(* IEC 61131-3 sources: brOscatLib/oscatNetw (part 7) *)

(* ---- TN_INPUT_MENU_POPUP.st ---- *)
FUNCTION_BLOCK TN_INPUT_MENU_POPUP
    (*http://www.oscat.de/images/OSCATNetwork/oscat_netlib121_en.pdf#page=178*)
    (* sicherstellen das rechteck immer innerhalb screen positioniert wird *)

    IF (XUS_TN_MENU_POPUP.bo_Activ = FALSE) AND (XUS_TN_MENU_POPUP.bo_Create = TRUE) THEN
    	XUS_TN_MENU_POPUP.bo_Activ := TRUE;
    	XUS_TN_MENU_POPUP.bo_Create := FALSE;
    	XUS_TN_MENU_POPUP.bo_Destroy := FALSE;
    	XUS_TN_MENU_POPUP.bo_Update := TRUE;

      (* Sub-Menu-Texte *)

    	XUS_TN_MENU_POPUP.in_Menu_E_Count := ELEMENT_COUNT(SEP:=BYTE#35,ELEMENT:=XUS_TN_MENU_POPUP.st_Menu_Text);

    	(* Anzahl Zeilen (Sub-Menu-Texte) bestimmen *)
    	XUS_TN_MENU_POPUP.in_ROWS := XUS_TN_MENU_POPUP.in_Menu_E_Count;

    	(* längsten Sub-Menu-Text suchen *)
    	XUS_TN_MENU_POPUP.in_COLS := INT#00;

    	FOR in_Count := INT#01 TO XUS_TN_MENU_POPUP.in_ROWS DO;
    		XUS_TN_MENU_POPUP.in_COLS:=MAX(LEN(ELEMENT_GET(SEP:=BYTE#35,POS:=in_Count - 1,ELEMENT:=XUS_TN_MENU_POPUP.st_Menu_Text)),XUS_TN_MENU_POPUP.in_COLS);
    	END_FOR

    	(* Horizontale Position überprüfen und korrigieren *)
    	IF (XUS_TN_MENU_POPUP.in_X + XUS_TN_MENU_POPUP.in_COLS) > INT#75 THEN
    		XUS_TN_MENU_POPUP.in_X := INT#79 - XUS_TN_MENU_POPUP.in_COLS - INT#04;
    	END_IF

      (* Vertikale Position überprüfen und korrigieren *)
    	IF (XUS_TN_MENU_POPUP.in_Y + XUS_TN_MENU_POPUP.in_ROWS) > INT#21 THEN
    		XUS_TN_MENU_POPUP.in_Y := INT#23 - XUS_TN_MENU_POPUP.in_ROWS - INT#2;
    	END_IF

    	XUS_TN_SCREEN.bo_Modal_Dialog := TRUE;

    	(* Hintergrund sichern *)
    	FB_TN_SC_AREA_SAVE(	Iin_X1 := XUS_TN_MENU_POPUP.in_X,
    									Iin_Y1 := XUS_TN_MENU_POPUP.in_Y,
    									Iin_X2 := XUS_TN_MENU_POPUP.in_X + XUS_TN_MENU_POPUP.in_COLS + INT#04,
    									Iin_Y2 := XUS_TN_MENU_POPUP.in_Y + XUS_TN_MENU_POPUP.in_ROWS + INT#02,
    									XUS_TN_SCREEN := XUS_TN_SCREEN);

    	(* Rahmen für Submenu zeichnen *)
    	FB_TN_SC_BOX(	Iin_X1 := XUS_TN_MENU_POPUP.in_X,
    					Iin_Y1 := XUS_TN_MENU_POPUP.in_Y,
    					Iin_X2 := XUS_TN_MENU_POPUP.in_X + XUS_TN_MENU_POPUP.in_COLS + INT#03,
    					Iin_Y2 := XUS_TN_MENU_POPUP.in_Y + XUS_TN_MENU_POPUP.in_ROWS + INT#01,
    					Iby_FILL := BYTE#32, (* Füllung *)
    					Iin_BORDER := INT#01, (* Single-Line Border *)
    					Iby_ATTR := XUS_TN_MENU_POPUP.by_Attr_oF,
    					XUS_TN_SCREEN := XUS_TN_SCREEN);

    	(* Shadow für Submenu zeichnen *)
    	FB_TN_SC_ADD_SHADOW(Iin_X1 := XUS_TN_MENU_POPUP.in_X + INT#1,
    						Iin_Y1 := XUS_TN_MENU_POPUP.in_Y + INT#1,
    						Iin_X2 := XUS_TN_MENU_POPUP.in_X + XUS_TN_MENU_POPUP.in_COLS + INT#04,
    						Iin_Y2 := XUS_TN_MENU_POPUP.in_Y + XUS_TN_MENU_POPUP.in_ROWS + INT#02,
    						Iin_OPTION := INT#00,
    						XUS_TN_SCREEN := XUS_TN_SCREEN);

    	(* Parameter laden *)
    	in_COL := XUS_TN_MENU_POPUP.in_X;
    	in_ROW := XUS_TN_MENU_POPUP.in_Y;
    	in_ROWS := XUS_TN_MENU_POPUP.in_ROWS;
    	in_COLS := XUS_TN_MENU_POPUP.in_COLS;

    	(* Trennlinien zeichnen *)
    	in_COLS := in_COLS + INT#02; (* Text um 2 Zeichen verlängern *)

    	FOR in_Count := INT#01 TO XUS_TN_MENU_POPUP.in_Menu_E_Count DO;
    		in_ROW := in_ROW + INT#01;

    		IF ELEMENT_GET(SEP:=BYTE#35,POS:=in_Count - 1,ELEMENT:=XUS_TN_MENU_POPUP.st_Menu_Text) = '-' THEN

    			FB_TN_SC_LINE(	Iin_Y1 := in_ROW,
    							Iin_X1 := in_COL,
    							Iin_Y2 := in_ROW,
    							Iin_X2 := in_COL + in_COLS + INT#01,
    							Iby_ATTR := XUS_TN_MENU_POPUP.by_Attr_oF,
    							Iby_BORDER := BYTE#01,
    							XUS_TN_SCREEN := XUS_TN_SCREEN);
    		END_IF
    	END_FOR
    END_IF

    IF (XUS_TN_MENU_POPUP.bo_Activ = TRUE) THEN

    	CASE BYTE_TO_INT(XUS_TN_MENU_POPUP.by_Input_Exten_Code) OF

    	65: (* Cursor oben *)
    		in_Scroll_Offset := -1;
    		XUS_TN_MENU_POPUP.bo_Update := TRUE;

    	66: (* Cursor unten *)
    		in_Scroll_Offset := 1;
    		XUS_TN_MENU_POPUP.bo_Update := TRUE;

    	13:  (* Enter *)
    		XUS_TN_MENU_POPUP.bo_Destroy := TRUE;

    	27:  (* Escape*)
    		XUS_TN_MENU_POPUP.bo_Destroy := TRUE;
    		XUS_TN_MENU_POPUP.in_Cur_Item := INT#00;

    	67..68: (* Cursor links oder rechts *)
    		XUS_TN_MENU_POPUP.bo_Destroy := TRUE;
    		XUS_TN_MENU_POPUP.in_Cur_Item := INT#00;

    	END_CASE
    END_IF

    (* POPUP-Menu updaten *)
    IF (XUS_TN_MENU_POPUP.bo_Activ = TRUE) AND (XUS_TN_MENU_POPUP.bo_Update = TRUE) THEN

    	XUS_TN_MENU_POPUP.bo_Update := FALSE;

    	(* überprüfung + nächstes anwählbares Sub-Menu suchen *)
    	in_index := XUS_TN_MENU_POPUP.in_Cur_Item;

    	IF (in_index < INT#01) OR (in_index > XUS_TN_MENU_POPUP.in_Menu_E_Count) THEN
    		in_Scroll_Offset := INT#01;
    		in_index := XUS_TN_MENU_POPUP.in_Menu_E_Count;
    	END_IF

    	(* aktueller Index steht auf Trennzeichen -> ändern *)
    	IF ELEMENT_GET(SEP:=BYTE#35,POS:=in_index-1,ELEMENT:=XUS_TN_MENU_POPUP.st_Menu_Text) = '-' THEN
    		in_Scroll_Offset := INT#01;
    	END_IF

    	(* Scroll-Offset *)
    	IF in_Scroll_Offset <> INT#00 THEN

    		FOR in_Count := INT#01 TO XUS_TN_MENU_POPUP.in_Menu_E_Count DO;

    			in_index:=INC2(in_index,in_Scroll_Offset,1,XUS_TN_MENU_POPUP.in_Menu_E_Count);

    			IF ELEMENT_GET(SEP:=BYTE#35,POS:=in_index - 1,ELEMENT:=XUS_TN_MENU_POPUP.st_Menu_Text) <> '-' THEN
    				EXIT;
    			END_IF

    		END_FOR
    	END_IF

    	XUS_TN_MENU_POPUP.in_Cur_Item := in_index;
    	in_Scroll_Offset := INT#00;

    	(* Parameter laden *)
    	in_COL  := XUS_TN_MENU_POPUP.in_X;
    	in_ROW  := XUS_TN_MENU_POPUP.in_Y;
    	in_ROWS := XUS_TN_MENU_POPUP.in_ROWS;
    	in_COLS := XUS_TN_MENU_POPUP.in_COLS;

    	(* SUB-MENU-Titel ausgeben *)
    	in_COLS := in_COLS + INT#02; (* Text um 2 Zeichen verlängern *)

    	FOR in_Count := INT#01 TO XUS_TN_MENU_POPUP.in_Menu_E_Count DO;

    		in_ROW := in_ROW + INT#01;

    		(* Zeichenfarbe bestimmen *)
    		IF in_Count = XUS_TN_MENU_POPUP.in_Cur_Item THEN
    			by_ATTR := XUS_TN_MENU_POPUP.by_Attr_mF;
    		ELSE
    			by_ATTR := XUS_TN_MENU_POPUP.by_Attr_oF;
    		END_IF

    		FB_TN_SC_WRITE_C.Ist_STRING := ELEMENT_GET(SEP:=BYTE#35,POS:=in_Count - 1,ELEMENT:=XUS_TN_MENU_POPUP.st_Menu_Text);

    		IF FB_TN_SC_WRITE_C.Ist_STRING <> '-' THEN

    			FB_TN_SC_WRITE_C(	Iin_Y := in_ROW,
    								Iin_X := in_COL + INT#01,
    								Iby_ATTR := by_ATTR,
    								Iin_LENGTH := in_COLS,
    								Iin_OPTION := INT#02, (* Center *)
    								XUS_TN_SCREEN := XUS_TN_SCREEN);
    		END_IF
    	END_FOR
    END_IF

    (* POPUP-Menu entfernen (Destroy) *)
    IF (XUS_TN_MENU_POPUP.bo_Activ = TRUE) AND (XUS_TN_MENU_POPUP.bo_Destroy = TRUE) THEN

    	XUS_TN_MENU_POPUP.bo_Destroy := FALSE;
    	XUS_TN_MENU_POPUP.bo_Activ := FALSE;

    	(* alten Hintergrund aus Speicher wiederherstellen *)
    	FB_TN_SC_AREA_RESTORE(XUS_TN_SCREEN := XUS_TN_SCREEN);

    	XUS_TN_SCREEN.bo_Modal_Dialog := FALSE;
    END_IF

    (* revision history

    ks	06. apr. 2011	rev 1.1
    	list_len und list_get durch element_count und element_get ersetzt

    ks	10. mai. 2010	rev 1.0
    	original version
    *)
END_FUNCTION_BLOCK

(* ---- TN_INPUT_SELECT_POPUP.st ---- *)
FUNCTION_BLOCK TN_INPUT_SELECT_POPUP
    (*http://www.oscat.de/images/OSCATNetwork/oscat_netlib121_en.pdf#page=178*)
    (* Benutzereingabe auswerten -> Selektion Text n *)
    IF (XUS_TN_INPUT_CONTROL_DATA.bo_Focus = TRUE) THEN

    	by_Cur_Key := XUS_TN_INPUT_CONTROL_DATA.by_Input_Exten_Code;

    	IF (us_TN_MENU_POPUP.bo_Activ = FALSE) THEN
    		us_TN_MENU_POPUP.by_Input_Exten_Code := BYTE#00;

    		(* Return-Taste auswerten *)
    		IF (by_Cur_Key = BYTE#13) THEN
    			(* Popup-Menu parameter übergeben *)
    			us_TN_MENU_POPUP.in_Y := XUS_TN_INPUT_CONTROL_DATA.in_Y;
    			us_TN_MENU_POPUP.in_X := XUS_TN_INPUT_CONTROL_DATA.in_X;
    			us_TN_MENU_POPUP.by_Attr_mF := XUS_TN_INPUT_CONTROL_DATA.by_Attr_mF;
    			us_TN_MENU_POPUP.by_Attr_oF := XUS_TN_INPUT_CONTROL_DATA.by_Attr_oF;
    			us_TN_MENU_POPUP.st_Menu_Text := XUS_TN_INPUT_CONTROL_DATA.st_Input_Data;
    			us_TN_MENU_POPUP.bo_Create := TRUE;
    			us_TN_MENU_POPUP.in_Cur_Item := INT#00;
    		END_IF

    		IF (us_TN_MENU_POPUP.in_Cur_Item > INT#00) THEN
    			XUS_TN_INPUT_CONTROL_DATA.in_selected := us_TN_MENU_POPUP.in_Cur_Item;
    			XUS_TN_INPUT_CONTROL_DATA.bo_Input_Entered := TRUE;
    			XUS_TN_INPUT_CONTROL_DATA.bo_Update_Input := TRUE;
    			us_TN_MENU_POPUP.in_Cur_Item := INT#00;
    		END_IF

    	ELSE
    		us_TN_MENU_POPUP.by_Input_Exten_Code := by_Cur_Key;
    	END_IF

    	(* Popup-Menu zyklisch aufrufen *)
    	FB_TN_INPUT_MENU_POPUP(Xus_TN_MENU_POPUP := us_TN_MENU_POPUP, XUS_TN_SCREEN := XUS_TN_SCREEN);

    END_IF

    (* Aktualisierung der Anzeige *)
    IF (XUS_TN_INPUT_CONTROL_DATA.bo_Update_Input = TRUE) OR (XUS_TN_INPUT_CONTROL_DATA.bo_Update_All = TRUE) THEN

    	(* Title-Text ausgeben *)
    	IF XUS_TN_INPUT_CONTROL_DATA.bo_Update_All = TRUE THEN

    		IF (XUS_TN_INPUT_CONTROL_DATA.in_Title_X_Offset = INT#00) AND (XUS_TN_INPUT_CONTROL_DATA.in_Title_Y_Offset = INT#00) THEN
    			(* wenn Offset X,Y =0 dann Titlestring links vom Element positionieren *)
    			FB_TN_SC_WRITE.Iin_Y := XUS_TN_INPUT_CONTROL_DATA.in_Y;
    			FB_TN_SC_WRITE.Iin_X := XUS_TN_INPUT_CONTROL_DATA.in_X - LEN(XUS_TN_INPUT_CONTROL_DATA.st_Title_String);

    		ELSE
    			(* Title-Text durch Row, Color-Offset ausgeben *)
    			FB_TN_SC_WRITE.Iin_Y := XUS_TN_INPUT_CONTROL_DATA.in_Y + XUS_TN_INPUT_CONTROL_DATA.in_Title_Y_Offset;
    			FB_TN_SC_WRITE.Iin_X := XUS_TN_INPUT_CONTROL_DATA.in_X + XUS_TN_INPUT_CONTROL_DATA.in_Title_X_Offset;
    		END_IF

    		(* Title-Text durch Row, Color-Offset ausgeben *)
    		FB_TN_SC_WRITE(	Iby_ATTR := XUS_TN_INPUT_CONTROL_DATA.by_Title_Attr,
    						Ist_STRING := XUS_TN_INPUT_CONTROL_DATA.st_Title_String,
    						XUS_TN_SCREEN := XUS_TN_SCREEN);
    	END_IF

    	in_Element_Count := ELEMENT_COUNT(SEP:=BYTE#35,ELEMENT:=XUS_TN_INPUT_CONTROL_DATA.st_Input_Data);

    	IF in_Element_Count > INT#00 THEN

    		XUS_TN_INPUT_CONTROL_DATA.in_selected:=LIMIT(1,XUS_TN_INPUT_CONTROL_DATA.in_selected,in_Element_Count);

    		in_index := XUS_TN_INPUT_CONTROL_DATA.in_selected;

    		st_String := ELEMENT_GET(SEP:=BYTE#35,POS:=in_index - 1,ELEMENT:=XUS_TN_INPUT_CONTROL_DATA.st_Input_Data);

    		st_String:= FIX(str:=st_String,
    						L:=LEN(XUS_TN_INPUT_CONTROL_DATA.st_Input_Mask),
    						C:=BYTE#32,
    						M:=XUS_TN_INPUT_CONTROL_DATA.in_Input_Option);

    		XUS_TN_INPUT_CONTROL_DATA.st_Input_String := st_String;

    		IF XUS_TN_INPUT_CONTROL_DATA.bo_Focus = TRUE THEN
    			by_Attr := XUS_TN_INPUT_CONTROL_DATA.by_Attr_mF;
    		ELSE
    			by_Attr := XUS_TN_INPUT_CONTROL_DATA.by_Attr_oF;
    		END_IF

    		FB_TN_SC_WRITE(	Iin_X := XUS_TN_INPUT_CONTROL_DATA.in_X,
    								Iin_Y := XUS_TN_INPUT_CONTROL_DATA.in_Y,
    								Iby_ATTR := by_Attr,
    								Ist_STRING := st_String,
    								XUS_TN_SCREEN := XUS_TN_SCREEN );
    	END_IF

    	(* Cursor auf aktuelle Position setzen *)
    	XUS_TN_INPUT_CONTROL_DATA.in_Cursor_X := XUS_TN_INPUT_CONTROL_DATA.in_X;
    	XUS_TN_INPUT_CONTROL_DATA.in_Cursor_Y := XUS_TN_INPUT_CONTROL_DATA.in_Y;

    	(* Update-Flag's rücksetzen *)
    	XUS_TN_INPUT_CONTROL_DATA.bo_Update_All   := FALSE;
    	XUS_TN_INPUT_CONTROL_DATA.bo_Update_Input := FALSE;

    END_IF

    (* revision history

    ks	06. apr. 2011	rev 1.1
    	list_len und list_get durch element_count und element_get ersetzt

    ks	10. mai. 2010	rev 1.0
    	original version
    *)
END_FUNCTION_BLOCK

(* ---- TN_INPUT_SELECT_TEXT.st ---- *)
FUNCTION_BLOCK TN_INPUT_SELECT_TEXT
    (*http://www.oscat.de/images/OSCATNetwork/oscat_netlib121_en.pdf#page=180*)
    (* Benutzereingabe auswerten -> Selektion Text n *)
    IF XUS_TN_INPUT_CONTROL_DATA.bo_Focus = TRUE THEN

    (* Leertaste-Taste auswerten *)
    	IF XUS_TN_INPUT_CONTROL_DATA.by_Input_ASCII_Code = BYTE#32 THEN
    		XUS_TN_INPUT_CONTROL_DATA.in_selected := XUS_TN_INPUT_CONTROL_DATA.in_selected + INT#01;
    		XUS_TN_INPUT_CONTROL_DATA.bo_Update_Input := TRUE;
    	END_IF

    	(* Return-Taste auswerten *)
    	IF XUS_TN_INPUT_CONTROL_DATA.by_Input_Exten_Code = BYTE#13 THEN
    		XUS_TN_INPUT_CONTROL_DATA.bo_Input_Entered := TRUE;
    	END_IF

    END_IF

    (* Aktualisierung der Anzeige *)
    IF (XUS_TN_INPUT_CONTROL_DATA.bo_Update_Input = TRUE) OR (XUS_TN_INPUT_CONTROL_DATA.bo_Update_All = TRUE) THEN

    	(* Title-Text ausgeben *)
    	IF XUS_TN_INPUT_CONTROL_DATA.bo_Update_All = TRUE THEN

    		IF (XUS_TN_INPUT_CONTROL_DATA.in_Title_X_Offset = INT#00) AND (XUS_TN_INPUT_CONTROL_DATA.in_Title_Y_Offset = INT#00) THEN
    			(* wenn Offset X,Y =0 dann Titlestring links vom Element positionieren *)
    			FB_TN_SC_WRITE.Iin_Y := XUS_TN_INPUT_CONTROL_DATA.in_Y;
    			FB_TN_SC_WRITE.Iin_X := XUS_TN_INPUT_CONTROL_DATA.in_X - LEN(XUS_TN_INPUT_CONTROL_DATA.st_Title_String);

    		ELSE
    			(* Title-Text durch Row, Color-Offset ausgeben *)
    			FB_TN_SC_WRITE.Iin_Y := XUS_TN_INPUT_CONTROL_DATA.in_Y + XUS_TN_INPUT_CONTROL_DATA.in_Title_Y_Offset;
    			FB_TN_SC_WRITE.Iin_X := XUS_TN_INPUT_CONTROL_DATA.in_X + XUS_TN_INPUT_CONTROL_DATA.in_Title_X_Offset;
    		END_IF

    		(* Title-Text durch Row, Color-Offset ausgeben *)
    		FB_TN_SC_WRITE(	Iby_ATTR := XUS_TN_INPUT_CONTROL_DATA.by_Title_Attr,
    						Ist_STRING := XUS_TN_INPUT_CONTROL_DATA.st_Title_String,
    						XUS_TN_SCREEN := XUS_TN_SCREEN);

    	END_IF

    	(* Eingabezeile verarbeiten *)

    	(* Anzahl der Elemente bestimmen *)
    	in_count := ELEMENT_COUNT(SEP:=BYTE#35,ELEMENT:=XUS_TN_INPUT_CONTROL_DATA.st_Input_Data);

    	IF in_count > INT#00 THEN

    		IF XUS_TN_INPUT_CONTROL_DATA.in_selected < INT#1 THEN
    			XUS_TN_INPUT_CONTROL_DATA.in_selected := INT#01;
    		END_IF

    		IF XUS_TN_INPUT_CONTROL_DATA.in_selected > in_count THEN
    			XUS_TN_INPUT_CONTROL_DATA.in_selected := INT#01;
    		END_IF

    		st_String := ELEMENT_GET(SEP:=BYTE#35,POS:=XUS_TN_INPUT_CONTROL_DATA.in_selected - 1,ELEMENT:=XUS_TN_INPUT_CONTROL_DATA.st_Input_Data);

    		st_String := FIX(	str:=st_String,
    							L:=LEN(XUS_TN_INPUT_CONTROL_DATA.st_Input_Mask),
    							C:=BYTE#32,
    							M:=XUS_TN_INPUT_CONTROL_DATA.in_Input_Option);

    		XUS_TN_INPUT_CONTROL_DATA.st_Input_String := st_String;

    		IF XUS_TN_INPUT_CONTROL_DATA.bo_Focus = TRUE THEN
    			by_Attr := XUS_TN_INPUT_CONTROL_DATA.by_Attr_mF;
    		ELSE
    			by_Attr := XUS_TN_INPUT_CONTROL_DATA.by_Attr_oF;
    		END_IF

    		FB_TN_SC_WRITE(	Iin_Y := XUS_TN_INPUT_CONTROL_DATA.in_Y,
    						Iin_X := XUS_TN_INPUT_CONTROL_DATA.in_X,
    						Iby_ATTR := by_Attr,
    						Ist_STRING := st_String,
    						XUS_TN_SCREEN := XUS_TN_SCREEN);
    	END_IF

    	(* Cursor auf aktuelle Position setzen *)
    	XUS_TN_INPUT_CONTROL_DATA.in_Cursor_Y := XUS_TN_INPUT_CONTROL_DATA.in_Y;
    	XUS_TN_INPUT_CONTROL_DATA.in_Cursor_X := XUS_TN_INPUT_CONTROL_DATA.in_X;

    	(* Update-Flag's rücksetzen *)
    	XUS_TN_INPUT_CONTROL_DATA.bo_Update_All := FALSE;
    	XUS_TN_INPUT_CONTROL_DATA.bo_Update_Input := FALSE;

    END_IF

    (* revision history

    ks	06. apr. 2011	rev 1.1
    	list_len und list_get durch element_count und element_get ersetzt

    ks	10. mai. 2010	rev 1.0
    	original version
    *)
END_FUNCTION_BLOCK

(* ---- TN_RECEIVE.st ---- *)
FUNCTION_BLOCK TN_RECEIVE
    (*http://www.oscat.de/images/OSCATNetwork/oscat_netlib121_en.pdf#page=182*)
    (* Datenempfang auswertung *)
    XUS_TN_SCREEN.by_Input_ASCII_Code := BYTE#00;
    XUS_TN_SCREEN.by_Input_Exten_Code := BYTE#00;

    IF R_BUF.SIZE > UINT#0 THEN
    	(* empfangene Daten auswerten *)
    	REQ_Size := R_BUF.SIZE;
    	REQ1 := R_BUF.BUFFER[0];
    	REQ2 := R_BUF.BUFFER[1];
    	REQ3 := R_BUF.BUFFER[2];

    	IF REQ1 = BYTE#27 AND REQ_Size >= UINT#3 THEN (* Escape *)
    		IF REQ2 = BYTE#91 THEN (* Cursor code *)
    			IF (REQ3 >= BYTE#65 AND REQ3 <= BYTE#68) OR (REQ3 = BYTE#72) OR (REQ3 = BYTE#75) THEN (* 65..68 = Cursor o,u,r,l / 72 = POS1 / 75 = ENDE *)
    				XUS_TN_SCREEN.by_Input_Exten_Code := REQ3;
    			END_IF
    		ELSIF REQ2 = BYTE#79 THEN (* Sondertasten F1/F2/F3/F4 *)
    			IF REQ3 >= BYTE#80 AND REQ3 <= BYTE#83 THEN
    				XUS_TN_SCREEN.by_Input_Exten_Code := REQ3;
    			END_IF
    		END_IF
    	ELSIF REQ1 >= BYTE#32 AND REQ1 <= BYTE#126 THEN
    		XUS_TN_SCREEN.by_Input_ASCII_Code := REQ1;
    		XUS_TN_SCREEN.bo_Input_ASCII_IsNum := ISC_NUM(REQ1); (* Auswertung auf Zahleneingabe *)
    	ELSIF REQ1 = BYTE#8 OR REQ1 = BYTE#9 OR REQ1 = BYTE#13 OR REQ1 = BYTE#27 THEN (* prüfe auf Steuerzeichen 8=Backspace / 9=Tabulator / 13=Return / 27=Escape *)
    		XUS_TN_SCREEN.by_Input_Exten_Code := REQ1;
    	END_IF

    	(* Empfangsbuffer Datenlänge null eintragen (Telegramm zerstören *)
    	R_BUF.SIZE := UINT#00;
    END_IF

    (* revision history
    ks	10. mai. 2010	rev 1.0
    	original version
    *)
END_FUNCTION_BLOCK

(* ---- TN_SC_ADD_SHADOW.st ---- *)
FUNCTION_BLOCK TN_SC_ADD_SHADOW
    (*http://www.oscat.de/images/OSCATNetwork/oscat_netlib121_en.pdf#page=184*)
    IF TN_SC_XY2_ERROR(IIN_X1,IIN_Y1,IIN_X2,IIN_Y2) THEN RETURN; END_IF

    IF IIN_Y1 < 0 OR IIN_X1 < 0 OR IIN_Y2 < 0 OR IIN_X2 < 0 THEN RETURN; END_IF (* min werte prüfen *)
    IF IIN_Y1 > 23 OR IIN_X1 > 79 OR IIN_Y2 > 23 OR IIN_X2 > 79 THEN RETURN; END_IF (* max werte prüfen *)

    in_Offset := (IIN_Y1 * 80) + IIN_X2;

    IF IIN_OPTION = INT#00 THEN
    	(* Schatten durch Farbanpassung erzeugen *)
    	FOR in_Y := IIN_Y1 TO IIN_Y2 DO
    		XUS_TN_SCREEN.bya_COLOR[in_Offset] := TN_SC_SHADOW_ATTR(XUS_TN_SCREEN.bya_COLOR[in_Offset]);
    		in_Offset := in_Offset + 80;
    		XUS_TN_SCREEN.bya_Line_Update[in_Y] := TRUE; (* Zeile für Update eintragen *)
    	END_FOR
    ELSE
    	(* Schatten durch Farbe Schwarz und Leerzeichen erzeugen *)
    	FOR in_Y := IIN_Y1 TO IIN_Y2 DO
    		XUS_TN_SCREEN.bya_COLOR[in_Offset] := BYTE#00;
    		XUS_TN_SCREEN.bya_CHAR[in_Offset] := BYTE#32;
    		in_Offset := in_Offset + 80;
    		XUS_TN_SCREEN.bya_Line_Update[in_Y] := TRUE; (* Zeile für Update eintragen *)
    	END_FOR
    END_IF

    in_Offset := (IIN_Y2 * 80) + IIN_X1;

    IF IIN_OPTION = INT#00 THEN
    	(* Schatten durch Farbanpassung erzeugen *)
    	FOR in_X  := IIN_X1 TO IIN_X2 DO
    		XUS_TN_SCREEN.bya_COLOR[in_Offset] := TN_SC_SHADOW_ATTR(XUS_TN_SCREEN.bya_COLOR[in_Offset]);
    		in_Offset := in_Offset + 1;
    	END_FOR
    ELSE
    	(* Schatten durch Farbe Schwarz und Leerzeichen erzeugen *)
    	FOR in_X  := IIN_X1 TO IIN_X2 DO
    		XUS_TN_SCREEN.bya_COLOR[in_Offset] := BYTE#00;
    		XUS_TN_SCREEN.bya_CHAR[in_Offset] := BYTE#32;
    		in_Offset := in_Offset + 1;
    	END_FOR
    END_IF

    (* revision history
    ks	10. mai. 2010	rev 1.0
    	original version
    *)
END_FUNCTION_BLOCK

(* ---- TN_SC_AREA_RESTORE.st ---- *)
FUNCTION_BLOCK TN_SC_AREA_RESTORE
    (*http://www.oscat.de/images/OSCATNetwork/oscat_netlib121_en.pdf#page=184*)
    IF XUS_TN_SCREEN.bya_BACKUP[0] > BYTE#00 THEN

    	(* Parameter auslesen *)
    	in_X1 := BYTE_TO_INT(XUS_TN_SCREEN.bya_BACKUP[1]);
    	in_Y1 := BYTE_TO_INT(XUS_TN_SCREEN.bya_BACKUP[2]);
    	in_X2 := BYTE_TO_INT(XUS_TN_SCREEN.bya_BACKUP[3]);
    	in_Y2 := BYTE_TO_INT(XUS_TN_SCREEN.bya_BACKUP[4]);

    	IF TN_SC_XY2_ERROR(in_X1,in_Y1,in_X2,in_Y2) THEN RETURN; END_IF
    	in_Offset_2 := 5;

    	(* CHAR und COLOR von BUFFER wiederherstellen *)
    	FOR in_Y := in_Y1 TO in_Y2 DO

    		XUS_TN_SCREEN.bya_Line_Update[in_Y] := TRUE; (* Zeile zum Updaten freigeben *)
    		in_Offset_1 := (in_Y * 80) + in_X1;

    		FOR in_X := in_X1 TO in_X2 DO

    			XUS_TN_SCREEN.bya_CHAR[in_Offset_1] := XUS_TN_SCREEN.bya_BACKUP[in_Offset_2];
    			in_Offset_2 := in_Offset_2 + INT#01;

    			XUS_TN_SCREEN.bya_COLOR[in_Offset_1] := XUS_TN_SCREEN.bya_BACKUP[in_Offset_2];
    			in_Offset_2 := in_Offset_2 + INT#01;
    			in_Offset_1 := in_Offset_1 + INT#01;

    		END_FOR
    	END_FOR

    	(* Daten als ungültig markieren *)
    	XUS_TN_SCREEN.bya_BACKUP[0] := BYTE#00;
    END_IF

    (* revision history
    ks	10. mai. 2010	rev 1.0
    	original version
    *)
END_FUNCTION_BLOCK

(* ---- TN_SC_AREA_SAVE.st ---- *)
FUNCTION_BLOCK TN_SC_AREA_SAVE
    (*http://www.oscat.de/images/OSCATNetwork/oscat_netlib121_en.pdf#page=185*)
    IF TN_SC_XY2_ERROR(IIN_X1,IIN_Y1,IIN_X2,IIN_Y2) THEN RETURN; END_IF

    (* Parameter ablegen *)
    XUS_TN_SCREEN.bya_BACKUP[0] := BYTE#1;
    XUS_TN_SCREEN.bya_BACKUP[1] := INT_TO_BYTE(IIN_X1);
    XUS_TN_SCREEN.bya_BACKUP[2] := INT_TO_BYTE(IIN_Y1);
    XUS_TN_SCREEN.bya_BACKUP[3] := INT_TO_BYTE(IIN_X2);
    XUS_TN_SCREEN.bya_BACKUP[4] := INT_TO_BYTE(IIN_Y2);

    in_Offset_2 := 5;
    (* CHAR und COLOR in BUFFER sichern *)
    FOR in_Y := IIN_Y1 TO IIN_Y2 DO

    	in_Offset_1 := (in_Y * 80) + IIN_X1;
    	FOR in_X := IIN_X1 TO IIN_X2 DO
    		XUS_TN_SCREEN.bya_BACKUP[in_Offset_2] := XUS_TN_SCREEN.bya_CHAR[in_Offset_1];
    		in_Offset_2 := in_Offset_2 + INT#01;
    		XUS_TN_SCREEN.bya_BACKUP[in_Offset_2] := XUS_TN_SCREEN.bya_COLOR[in_Offset_1];
    		in_Offset_2 := in_Offset_2 + INT#01;
    		in_Offset_1 := in_Offset_1 + INT#01;
    	END_FOR
    END_FOR

    (* revision history
    ks	10. mai. 2010	rev 1.0
    	original version
    *)
END_FUNCTION_BLOCK

(* ---- TN_SC_BOX.st ---- *)
FUNCTION_BLOCK TN_SC_BOX
    (*http://www.oscat.de/images/OSCATNetwork/oscat_netlib121_en.pdf#page=186*)
    IF TN_SC_XY2_ERROR(IIN_X1,IIN_Y1,IIN_X2,IIN_Y2) THEN RETURN; END_IF

    (* Bordertype bestimmen *)
    CASE IIN_BORDER OF
    0:
    	in_Border_Offset := 0;
    1:
    	by_BorderChar_L_T := BYTE#218; (* links oben *)
    	by_BorderChar_T := BYTE#196; (* oben *)
    	by_BorderChar_R_T := BYTE#191; (* rechts oben *)
    	by_BorderChar_L := BYTE#179; (* links *)
    	by_BorderChar_R := BYTE#179; (* rechts *)
    	by_BorderChar_B := BYTE#196; (* unten *)
    	by_BorderChar_L_B := BYTE#217; (* links unten *)
    	by_BorderChar_R_B := BYTE#192; (* rechts unten *)
    	in_Border_Offset := 1;
     2:
    	by_BorderChar_L_T := BYTE#201;
    	by_BorderChar_T := BYTE#205;
    	by_BorderChar_R_T := BYTE#187;
    	by_BorderChar_L := BYTE#186;
    	by_BorderChar_R := BYTE#186;
    	by_BorderChar_B := BYTE#205;
    	by_BorderChar_L_B := BYTE#188;
    	by_BorderChar_R_B := BYTE#200;
    	in_Border_Offset := 1;
    ELSE
    	by_BorderChar_L_T := BYTE#32;
    	by_BorderChar_T := BYTE#32;
    	by_BorderChar_R_T := BYTE#32;
    	by_BorderChar_L := BYTE#32;
    	by_BorderChar_R := BYTE#32;
    	by_BorderChar_B := BYTE#32;
    	by_BorderChar_L_B := BYTE#32;
    	by_BorderChar_R_B := BYTE#32;
    	in_Border_Offset := 1;

    END_CASE

    IF IBY_FILL > BYTE#0 THEN (* FILL Zeichen vorhanden ? -> Box zeichnen *)

    	(* Fill-Function um eine Zeichenreihe kleiner zeichnen *)
    	FB_TN_SC_FILL(	IIN_Y1 := IIN_Y1 + in_Border_Offset,
    					IIN_X1 := IIN_X1 + in_Border_Offset,
    					IIN_Y2 := IIN_Y2 - in_Border_Offset,
    					IIN_X2 := IIN_X2 - in_Border_Offset,
    					Iby_CHAR := IBY_FILL,
    					IBY_ATTR := IBY_ATTR,
    					XUS_TN_SCREEN := XUS_TN_SCREEN);
    END_IF

    IF IIN_BORDER = 0 THEN RETURN; END_IF

    (* linken und rechten Rand ausgeben *)

    in_Offset_1 := (IIN_Y1 * 80) + IIN_X1;
    in_Offset_2 := (IIN_Y1 * 80) + IIN_X2;

    FOR in_Y := IIN_Y1 TO IIN_Y2 DO

    	(* Zeile zum Updaten freigeben *)
    	XUS_TN_SCREEN.bya_Line_Update[in_Y] := TRUE;

    	XUS_TN_SCREEN.bya_CHAR[in_Offset_1] := by_BorderChar_L;
    	XUS_TN_SCREEN.bya_COLOR[in_Offset_1] := IBY_ATTR;

    	XUS_TN_SCREEN.bya_CHAR[in_Offset_2] := by_BorderChar_R;
    	XUS_TN_SCREEN.bya_COLOR[in_Offset_2] := IBY_ATTR;

    	in_Offset_1 := in_Offset_1 + 80;
    	in_Offset_2 := in_Offset_2 + 80;

    END_FOR

    (* unteren und oberen Rand ausgeben *)
    in_Offset_1 := (IIN_Y1 * 80) + IIN_X1;
    in_Offset_2 := (IIN_Y2 * 80) + IIN_X1;

    FOR in_X := IIN_X1 TO IIN_X2 DO

    	XUS_TN_SCREEN.bya_CHAR[in_Offset_1] := by_BorderChar_T;
    	XUS_TN_SCREEN.bya_COLOR[in_Offset_1] := IBY_ATTR;

    	XUS_TN_SCREEN.bya_CHAR[in_Offset_2] := by_BorderChar_B;
    	XUS_TN_SCREEN.bya_COLOR[in_Offset_2] := IBY_ATTR;

    	in_Offset_1 := in_Offset_1 + INT#1;
    	in_Offset_2 := in_Offset_2 + INT#1;

    END_FOR

    (* linke obere Ecke ausgeben *)
    in_Offset_1 := (IIN_Y1 * 80) + IIN_X1;
    XUS_TN_SCREEN.bya_CHAR[in_Offset_1] := by_BorderChar_L_T;
    XUS_TN_SCREEN.bya_COLOR[in_Offset_1] := IBY_ATTR;

    (* rechte obere Ecke ausgeben *)
    in_Offset_1 := (IIN_Y1 * 80) + IIN_X2;
    XUS_TN_SCREEN.bya_CHAR[in_Offset_1] := by_BorderChar_R_T;
    XUS_TN_SCREEN.bya_COLOR[in_Offset_1] := IBY_ATTR;

    (* linke untere Ecke ausgeben *)
    in_Offset_1 := (IIN_Y2 * 80) + IIN_X1;
    XUS_TN_SCREEN.bya_CHAR[in_Offset_1] := by_BorderChar_R_B;
    XUS_TN_SCREEN.bya_COLOR[in_Offset_1] := IBY_ATTR;

    (* rechte untere Ecke ausgeben *)
    in_Offset_1 := (IIN_Y2 * 80) + IIN_X2;
    XUS_TN_SCREEN.bya_CHAR[in_Offset_1] := by_BorderChar_L_B;
    XUS_TN_SCREEN.bya_COLOR[in_Offset_1] := IBY_ATTR;

    (* revision history
    ks	10. mai. 2010	rev 1.0
    	original version
    *)
END_FUNCTION_BLOCK

(* ---- TN_SC_FILL.st ---- *)
FUNCTION_BLOCK TN_SC_FILL
    (*http://www.oscat.de/images/OSCATNetwork/oscat_netlib121_en.pdf#page=187*)
    IF TN_SC_XY2_ERROR(IIN_X1,IIN_Y1,IIN_X2,IIN_Y2) THEN RETURN; END_IF

    FOR in_Y := IIN_Y1 TO IIN_Y2 DO
    	XUS_TN_SCREEN.bya_Line_Update[in_Y] := TRUE; (* Zeile zum Updaten freigeben *)
    	in_Offset := (in_Y * 80) + IIN_X1;
    	FOR in_X := IIN_X1 TO IIN_X2 DO
    		XUS_TN_SCREEN.bya_CHAR[in_Offset]  := IBY_CHAR; (* Zeichen eintragen *)
    		XUS_TN_SCREEN.bya_COLOR[in_Offset] := IBY_ATTR; (* Farbe eintragen *)
    		in_Offset := in_Offset + 1;
    	END_FOR
    END_FOR

    (* revision history
    ks	10. mai. 2010	rev 1.0
    	original version
    *)
END_FUNCTION_BLOCK

(* ---- TN_SC_LINE.st ---- *)
FUNCTION_BLOCK TN_SC_LINE
    (*http://www.oscat.de/images/OSCATNetwork/oscat_netlib121_en.pdf#page=188*)
    IF TN_SC_XY2_ERROR(IIN_X1,IIN_Y1,IIN_X2,IIN_Y2) THEN RETURN; END_IF

    (* Bordertype bestimmen *)
    IF IBY_BORDER = BYTE#01 THEN (* Single Line *)
    	by_Connect_Top_Char := BYTE#16#C2;
    	by_Connect_Bottom_Char := BYTE#16#C1;
    	by_Connect_Left_Char := BYTE#16#C3;
    	by_Connect_Right_Char := BYTE#16#B4;
    	by_Horzontal_Line_Char := BYTE#16#C4;
    	by_Vertikal_Line_Char := BYTE#16#B3;
    	by_Connect_Cruz_Char := BYTE#16#C5;
    ELSIF IBY_BORDER = BYTE#02 THEN	(* Double Linie *)
    	by_Connect_Top_Char := BYTE#16#CB;
    	by_Connect_Bottom_Char := BYTE#16#CA;
    	by_Connect_Left_Char := BYTE#16#CC;
    	by_Connect_Right_Char := BYTE#16#B9;
    	by_Horzontal_Line_Char := BYTE#16#CD;
    	by_Vertikal_Line_Char := BYTE#16#BA;
    	by_Connect_Cruz_Char := BYTE#16#CE;
    ELSE (* Full Linie *)
    	by_Connect_Top_Char := IBY_BORDER;
    	by_Connect_Bottom_Char := IBY_BORDER;
    	by_Connect_Left_Char := IBY_BORDER;
    	by_Connect_Right_Char := IBY_BORDER;
    	by_Horzontal_Line_Char := IBY_BORDER;
    	by_Vertikal_Line_Char := IBY_BORDER;
    	by_Connect_Cruz_Char := IBY_BORDER;
    END_IF

    (* Vertikale Linie zeichnen *)
    IF IIN_X1 = IIN_X2 THEN
    	in_Offset_1 := (IIN_Y1 * 80) + IIN_X1;
    	FOR in_ROW_Index := IIN_Y1 TO IIN_Y2 DO
    		by_old_Char := XUS_TN_SCREEN.bya_CHAR[in_Offset_1]; (* bestehendes Zeichen auslesen *)
    		by_Char := by_Vertikal_Line_Char; (* Standardzeichen vorbelegen *)
    		IF by_old_Char = by_Horzontal_Line_Char THEN (* Schnittpunkt erkannt *)
    			IF in_ROW_Index = IIN_Y1 THEN (* Anfang der Linie behandeln *)
    				by_Char := by_Connect_Top_Char;
    			ELSIF in_ROW_Index = IIN_Y2 THEN (* Ende der Linie behandeln *)
    				by_Char := by_Connect_Bottom_Char;
    			ELSE (* Kreuzungspunkt behandeln *)
    				by_Char := by_Connect_Cruz_Char;
    			END_IF
    		END_IF
    		XUS_TN_SCREEN.bya_Line_Update[in_ROW_Index] := TRUE; (* Zeile zum Updaten freigeben *)
    		XUS_TN_SCREEN.bya_CHAR[in_Offset_1] := by_Char;
    		XUS_TN_SCREEN.bya_COLOR[in_Offset_1] := IBY_ATTR;
    		in_Offset_1 := in_Offset_1 + 80;
    	END_FOR

    ELSIF IIN_Y1 = IIN_Y2 THEN (* Horzontale Linie zeichnen *)
    	XUS_TN_SCREEN.bya_Line_Update[IIN_Y1] := TRUE; (* Zeile zum Updaten freigeben *)
    	in_Offset_1 := (IIN_Y1 * 80) + IIN_X1;
    	FOR in_COL_Index := IIN_X1 TO IIN_X2 DO
    		by_old_Char := XUS_TN_SCREEN.bya_CHAR[in_Offset_1]; (* bestehendes Zeichen auslesen *)
    		by_Char := by_Horzontal_Line_Char; (* Standardzeichen vorbelegen *)
    		IF by_old_Char = by_Vertikal_Line_Char THEN (* Schnittpunkt erkannt *)
    			IF in_COL_Index = IIN_X1 THEN (* Anfang der Linie behandeln *)
    				by_Char := by_Connect_Left_Char;
    			ELSIF in_COL_Index = IIN_X2 THEN (* Ende der Linie behandeln *)
    				by_Char := by_Connect_Right_Char;
    			ELSE (* Kreuzungspunkt behandeln *)
    				by_Char := by_Connect_Cruz_Char;
    			END_IF
    		END_IF
    		XUS_TN_SCREEN.bya_CHAR[in_Offset_1] := by_Char;
    		XUS_TN_SCREEN.bya_COLOR[in_Offset_1] := IBY_ATTR;
    		in_Offset_1 := in_Offset_1 + 1;
    	END_FOR
    END_IF

    (* revision history
    ks	10. mai. 2010	rev 1.0
    	original version
    *)
END_FUNCTION_BLOCK

(* ---- TN_SC_READ_ATTR.st ---- *)
FUNCTION_BLOCK TN_SC_READ_ATTR
    (*http://www.oscat.de/images/OSCATNetwork/oscat_netlib121_en.pdf#page=190*)
    IF TN_SC_XY_ERROR(IIN_X,IIN_Y) THEN RETURN; END_IF
    in_Offset := (IIN_Y * 80) + IIN_X;
    OBY_ATTR := XUS_TN_SCREEN.bya_COLOR[in_Offset]; (* Attribute auslesen *)

    (* revision history
    ks	10. mai. 2010	rev 1.0
    	original version
    *)
END_FUNCTION_BLOCK

(* ---- TN_SC_READ_CHAR.st ---- *)
FUNCTION_BLOCK TN_SC_READ_CHAR
    (*http://www.oscat.de/images/OSCATNetwork/oscat_netlib121_en.pdf#page=190*)
    IF TN_SC_XY_ERROR(IIN_X,IIN_Y) THEN RETURN; END_IF
    in_Offset := (IIN_Y * 80) + IIN_X;
    OBY_CHAR := XUS_TN_SCREEN.bya_CHAR[in_Offset]; (* Charakter auslesen *)

    (* revision history
    ks	10. mai. 2010	rev 1.0
    	original version
    *)
END_FUNCTION_BLOCK

(* ---- TN_SC_VIEWPORT.st ---- *)
FUNCTION_BLOCK TN_SC_VIEWPORT
    (*http://www.oscat.de/images/OSCATNetwork/oscat_netlib121_en.pdf#page=191*)
    (* LOG-Messages ausgeben *)

    IF XUS_LOG_VIEWPORT.UPDATE AND FB_TON.Q THEN (* Update gewünscht und Verzögerungszeit abgelaufen *)
    	XUS_LOG_VIEWPORT.UPDATE := FALSE;
    	FOR in_count := 1 TO XUS_LOG_VIEWPORT.COUNT DO (* Alle Viewport-Zeilen abarbeiten *)
    		in_index := XUS_LOG_VIEWPORT.LINE_ARRAY[in_count];
    		(* Farbe aus den Option-Parameter auslesen >0,Level,Back,Front< *)
    		in_Color := DWORD_TO_INT(XUS_LOG_CONTROL.MSG_OPTION[in_index] AND DWORD#2#1111);

    		CASE in_Color OF
    		0..3: by_Attr := BYTE_OF_DWORD(IDW_ATTR_1,INT_TO_BYTE(in_Color));
    		4..7: by_Attr := BYTE_OF_DWORD(IDW_ATTR_2,INT_TO_BYTE(in_Color));
    		ELSE
    			by_Attr := BYTE_OF_DWORD(IDW_ATTR_1,BYTE#0);
    		END_CASE

    		(* Message (Text + Farbe) ausgeben *)
    		FB_TN_SC_WRITE(	IIN_Y := IIN_Y + in_count - INT#01,
    						IIN_X := IIN_X,
    						Iby_ATTR := by_Attr,
    						Ist_STRING := FIX(str := XUS_LOG_CONTROL.MSG[in_index], L := IIN_WIDTH, C := BYTE#32, M := INT#00), (* String rechts ergänzen bzw. kürzen *)
    						XUS_TN_SCREEN := XUS_TN_SCREEN);

    	END_FOR

    	(* Timer stoppen/rücksetzen *)
    	FB_TON.IN := FALSE;
    	FB_TON.PT := ITI_TIME;
    	FB_TON();

    END_IF

    (* Update-Zeitverzoegerung *)
    FB_TON.IN := TRUE;
    FB_TON.PT := ITI_TIME;
    FB_TON();

    (* revision history
    ks	10. mai. 2010	rev 1.0
    	original version
    *)
END_FUNCTION_BLOCK

(* ---- TN_SC_WRITE.st ---- *)
FUNCTION_BLOCK TN_SC_WRITE
    (*http://www.oscat.de/images/OSCATNetwork/oscat_netlib121_en.pdf#page=192*)
    in_String_Length := LEN(IST_STRING);
    IF TN_SC_XY_ERROR(IIN_X + in_String_Length - 1,IIN_Y) THEN RETURN; END_IF
    XUS_TN_SCREEN.bya_Line_Update[IIN_Y] := TRUE; (* Zeile zum Updaten freigeben *)
    in_Offset := (IIN_Y * 80) + IIN_X; (* Offset des ersten Zeichen berechnen *)
    bo_Color := IBY_ATTR <> BYTE#00;

    (* Zeichen und Attribute des String kopieren *)
    FOR in_Char_Index := 1 TO in_String_Length DO
    	IF bo_Color THEN XUS_TN_SCREEN.bya_COLOR[in_Offset] := IBY_ATTR; END_IF
    	XUS_TN_SCREEN.bya_CHAR[in_Offset] := CODE(STR:=IST_STRING,POS:=in_Char_Index);
    	in_Offset := in_Offset + INT#1;
    END_FOR

    XUS_TN_SCREEN.in_EOS_Offset := in_Offset; (* End of String Offset sichern *)

    (* revision history
    ks	10. mai. 2010	rev 1.0
    	original version
    *)
END_FUNCTION_BLOCK

(* ---- TN_SC_WRITE_ATTR.st ---- *)
FUNCTION_BLOCK TN_SC_WRITE_ATTR
    (*http://www.oscat.de/images/OSCATNetwork/oscat_netlib121_en.pdf#page=193*)
    IF TN_SC_XY_ERROR(IIN_X,IIN_Y) THEN RETURN; END_IF
    in_Offset := (IIN_Y * 80) + IIN_X;
    XUS_TN_SCREEN.bya_COLOR[in_Offset] := IBY_ATTR; (* Attribute schreiben *)

    (* revision history
    ks	10. mai. 2010	rev 1.0
    	original version
    *)
END_FUNCTION_BLOCK

(* ---- TN_SC_WRITE_C.st ---- *)
FUNCTION_BLOCK TN_SC_WRITE_C
    (*http://www.oscat.de/images/OSCATNetwork/oscat_netlib121_en.pdf#page=193*)
    (* Text ausgeben *)
    FB_TN_SC_WRITE( IIN_Y := IIN_Y,
    				IIN_X := IIN_X,
    				IBY_ATTR := IBY_ATTR,
    				IST_STRING := FIX(str:=IST_STRING,L:=IIN_LENGTH,C:=BYTE#32,M:=IIN_OPTION),
    				XUS_TN_SCREEN := XUS_TN_SCREEN);

    (* revision history
    ks	10. mai. 2010	rev 1.0
    	original version
    *)
END_FUNCTION_BLOCK

(* ---- TN_SC_WRITE_CHAR.st ---- *)
FUNCTION_BLOCK TN_SC_WRITE_CHAR
    (*http://www.oscat.de/images/OSCATNetwork/oscat_netlib121_en.pdf#page=194*)
    IF TN_SC_XY_ERROR(IIN_X,IIN_Y) THEN RETURN; END_IF
    in_Offset := (IIN_Y * 80) + IIN_X;
    XUS_TN_SCREEN.bya_CHAR[in_Offset] := IBY_CHAR; (* Charakter schreiben *)

    (* revision history
    ks	10. mai. 2010	rev 1.0
    	original version
    *)
END_FUNCTION_BLOCK

(* ---- TN_SC_WRITE_EOS.st ---- *)
FUNCTION_BLOCK TN_SC_WRITE_EOS
    (*http://www.oscat.de/images/OSCATNetwork/oscat_netlib121_en.pdf#page=195*)
    TN_SC_WRITE(Iin_Y := XUS_TN_SCREEN.in_EOS_Offset / 80, (* aktuelle Zeile ausrechnen *)
    			Iin_X := XUS_TN_SCREEN.in_EOS_Offset MOD 80, (* aktuelle Spalte ausrechnen *)
    			IBY_ATTR := IBY_ATTR,
    			IST_STRING := IST_STRING,
    			XUS_TN_SCREEN := XUS_TN_SCREEN);

    (* revision history
    ks	10. mai. 2010	rev 1.0
    	original version
    *)
END_FUNCTION_BLOCK

(* ---- TN_SEND_ROWS.st ---- *)
FUNCTION_BLOCK TN_SEND_ROWS
    (*http://www.oscat.de/images/OSCATNetwork/oscat_netlib121_en.pdf#page=183*)
    (* Verbindung vorhanden und kein Datensenden aktiv *)
    IF (IP_C.C_STATE < BYTE#127 OR S_BUF.SIZE > UINT#0) THEN
    	RETURN; (* nein -> Baustein beenden *)
    END_IF

    (* aktuellen Schreibindex laden *)
    in_Write_Index := UINT_TO_INT(S_BUF.SIZE) - 1;

    (* aktuellen Schreibindex zwischenspeichern *)
    in_Write_Index_Backup := in_Write_Index;

    (* positive Flanke Connect on *)
    IF (IP_C.C_STATE = BYTE#254) OR (XUS_TN_SCREEN.bo_Clear_Screen) THEN

    	(* Clear-Screen Meldung rücksetzen *)
    	XUS_TN_SCREEN.bo_Clear_Screen := FALSE;

    	(* alle Zeilen für Update markieren *)
    	FOR in_Line_Count := INT#00 TO INT#23 DO
    		XUS_TN_SCREEN.bya_Line_Update[in_Line_Count] := TRUE;
    	END_FOR

    	(* ESC [0;30,40m  Reset Attributes + Black,Black *)
    	in_Write_Index := in_Write_Index + INT#1;
    	S_BUF.BUFFER[in_Write_Index] := BYTE#16#1B; (* ESC *)
    	in_Write_Index := in_Write_Index + INT#1;
    	S_BUF.BUFFER[in_Write_Index] := BYTE#16#5B; (* [ *)
    	in_Write_Index := in_Write_Index + INT#1;
    	S_BUF.BUFFER[in_Write_Index] := BYTE#16#30; (* 0 *)
    	in_Write_Index := in_Write_Index + INT#1;
    	S_BUF.BUFFER[in_Write_Index] := BYTE#16#3B; (* ; *)
    	in_Write_Index := in_Write_Index + INT#1;
    	S_BUF.BUFFER[in_Write_Index] := BYTE#16#33; (* 3 *)

    	(* Einerstelle Farbe Foreground ausgeben *)
    	in_Write_Index := in_Write_Index + INT#1;
    	S_BUF.BUFFER[in_Write_Index] := (SHR(XUS_TN_SCREEN.by_Clear_Screen_Attr,4) OR BYTE#16#30);

    	in_Write_Index := in_Write_Index + INT#1;
    	S_BUF.BUFFER[in_Write_Index] := BYTE#16#3B; (* ; *)
    	in_Write_Index := in_Write_Index + INT#1;
    	S_BUF.BUFFER[in_Write_Index] := BYTE#16#34; (* 4 *)

    	(* Einerstelle Farbe Background ausgeben *)
    	in_Write_Index := in_Write_Index + INT#1;
    	S_BUF.BUFFER[in_Write_Index] := ((XUS_TN_SCREEN.by_Clear_Screen_Attr AND BYTE#16#07) OR BYTE#16#30);

    	in_Write_Index := in_Write_Index + INT#1;
    	S_BUF.BUFFER[in_Write_Index] := BYTE#16#6D; (* m *)

    	(* ESC[2J Clear screen and home cursor *)
    	in_Write_Index := in_Write_Index + INT#1;
    	S_BUF.BUFFER[in_Write_Index] := BYTE#16#1B; (* ESC *)
    	in_Write_Index := in_Write_Index + INT#1;
    	S_BUF.BUFFER[in_Write_Index] := BYTE#16#5B; (* [ *)
    	in_Write_Index := in_Write_Index + INT#1;
    	S_BUF.BUFFER[in_Write_Index] := BYTE#16#32; (* 2 *)
    	in_Write_Index := in_Write_Index + INT#1;
    	S_BUF.BUFFER[in_Write_Index] := BYTE#16#4A; (* J *)

    	(* ESC [?7l Off *)
    	in_Write_Index := in_Write_Index + INT#1;
    	S_BUF.BUFFER[in_Write_Index] := BYTE#16#1B; (* ESC *)
    	in_Write_Index := in_Write_Index + INT#1;
    	S_BUF.BUFFER[in_Write_Index] := BYTE#16#5B; (* [ *)
    	in_Write_Index := in_Write_Index + INT#1;
    	S_BUF.BUFFER[in_Write_Index] := BYTE#16#3F; (* ? *)
    	in_Write_Index := in_Write_Index + INT#1;
    	S_BUF.BUFFER[in_Write_Index] := BYTE#16#37; (* 7 *)
    	in_Write_Index := in_Write_Index + INT#1;
    	S_BUF.BUFFER[in_Write_Index] := BYTE#16#6C; (* l *)

    END_IF

    in_Last_Row_Index := INT#0;
    bo_Break_Loop := FALSE;
    in_Write_Stop := S_BUF_SIZE - 20;

    (* alle Zeilen durchlaufen *)
    FOR in_Line_Count := 0 TO 23 DO

    	in_Offset := in_Row_Count * INT#80;

    	(* prüfen ob Update einer Zeile notwendig ist bzw. nach Reconnect *)
    	IF (XUS_TN_SCREEN.bya_Line_Update[in_Row_Count] = TRUE) THEN

    		(* Schreib-Cursor positionieren *)
    		in_Write_Index := in_Write_Index + INT#1;
    		S_BUF.BUFFER[in_Write_Index] := BYTE#16#1B; (* ESC *)
    		in_Write_Index := in_Write_Index + INT#1;
    		S_BUF.BUFFER[in_Write_Index] := BYTE#16#5B; (* [ *)

    		(* Zehnerstelle Zeilennummer ausgeben *)
    		in_Write_Index := in_Write_Index + INT#1;
    		S_BUF.BUFFER[in_Write_Index] :=
    		SHR(INT_TO_BCDC(in_Row_Count + INT#1),INT#4) OR BYTE#16#30;

    		(* Einerstelle Zeilennummer ausgeben *)
    		in_Write_Index := in_Write_Index + INT#1;
    		S_BUF.BUFFER[in_Write_Index] :=
    		(INT_TO_BCDC(in_Row_Count + INT#1) AND BYTE#16#0F) OR BYTE#16#30;

    		in_Write_Index := in_Write_Index + INT#1;
    		S_BUF.BUFFER[in_Write_Index] := BYTE#16#3B; (* ; *)
    		in_Write_Index := in_Write_Index + INT#1;
    		S_BUF.BUFFER[in_Write_Index] := BYTE#16#31; (* 1 *)
    		in_Write_Index := in_Write_Index + INT#1;
    		S_BUF.BUFFER[in_Write_Index] := BYTE#16#48; (* H *)

    		(* alle Spalten einer Zeile durchlaufen *)
    		FOR in_Col_Count := 0 TO 79 DO

    			(* aktuelle Farbe bestimmen *)
    			by_Cur_Color := XUS_TN_SCREEN.bya_COLOR[in_Offset];
    			IF (by_Cur_Color <> by_last_Color) OR (in_Col_Count = INT#00) THEN

    				(* Farbeinstellung: ANSI-Sequenz ESC[X;Y;Zm ausgeben *)
    				in_Write_Index := in_Write_Index + INT#1;
    				S_BUF.BUFFER[in_Write_Index] := BYTE#16#1B; (* ESC *)

    				in_Write_Index := in_Write_Index + INT#1;
    				S_BUF.BUFFER[in_Write_Index] := BYTE#16#5B; (* [ *)

    				(* Farbeinstellung: dunkel oder Hell und blinken bestimmen *)

    					IF (((by_Cur_Color AND BYTE#2#10001000) XOR (by_last_Color AND BYTE#2#10001000)) <> BYTE#00) OR (in_Col_Count = 0) THEN

    						in_Write_Index := in_Write_Index + INT#1;
    						S_BUF.BUFFER[in_Write_Index] := BYTE#16#30; (* 0 *)
    						in_Write_Index := in_Write_Index + INT#1;
    						S_BUF.BUFFER[in_Write_Index] := BYTE#16#3B; (* ; *)

    						(* keine dunklen Farben gewünscht -> dann Bold & Bright *)
    						IF (by_Cur_Color AND BYTE#2#00001000) = BYTE#2#00000000 THEN

    							(* auf Bold & Btight Farben umstellen *)
    							in_Write_Index := in_Write_Index + INT#1;
    							S_BUF.BUFFER[in_Write_Index] := BYTE#16#31; (* 1 *)
    							in_Write_Index := in_Write_Index + INT#1;
    							S_BUF.BUFFER[in_Write_Index] := BYTE#16#3B; (* ; *)

    						END_IF

    						(* blinkenden Farben gewünscht *)
    						IF (by_Cur_Color AND BYTE#2#10000000) = BYTE#2#10000000 THEN

    							(* auf Bold & Bright Farben umstellen *)
    							in_Write_Index := in_Write_Index + INT#1;
    							S_BUF.BUFFER[in_Write_Index] := BYTE#16#35; (* 5 *)
    							in_Write_Index := in_Write_Index + INT#1;
    							S_BUF.BUFFER[in_Write_Index] := BYTE#16#3B; (* ; *)

    						END_IF

    					END_IF

    					(* Zehnerstelle Farbe Foreground ausgeben *)
    					in_Write_Index := in_Write_Index + INT#1;
    					S_BUF.BUFFER[in_Write_Index] := BYTE#16#33; (* 3 *)

    					(* Einerstelle Farbe Foreground ausgeben *)
    					in_Write_Index := in_Write_Index + INT#1;
    					S_BUF.BUFFER[in_Write_Index] := ((SHR(by_Cur_Color,4) AND BYTE#2#00000111) OR BYTE#16#30);

    					in_Write_Index := in_Write_Index + INT#1;
    					S_BUF.BUFFER[in_Write_Index] := BYTE#16#3B; (* ; *)

    					(* Zehnerstelle Farbe Background ausgeben *)
    					in_Write_Index := in_Write_Index + INT#1;
    					S_BUF.BUFFER[in_Write_Index] := BYTE#16#34; (* 4 *)

    					(* Einerstelle Farbe Background ausgeben *)
    					in_Write_Index := in_Write_Index + INT#1;
    					S_BUF.BUFFER[in_Write_Index] := ((by_Cur_Color AND BYTE#2#00000111) OR BYTE#16#30);

    					in_Write_Index := in_Write_Index + INT#1;
    					S_BUF.BUFFER[in_Write_Index] := BYTE#16#6D; (* m *)

    					(* neue Farbe als letzt verwendete speichern *)
    					by_last_Color := by_Cur_Color;

    				END_IF

    				(* Buffer Ende vorzeitig erreicht -> Ende *)
    				IF (in_Write_Index > in_Write_Stop) THEN

    					bo_Break_Loop := TRUE;
    					EXIT;

    				END_IF

    				(* ein TEXT-Zeichen von Screenbuffer in den Sendebuffer übertragen *)
    				in_Write_Index := in_Write_Index + INT#1;
    				S_BUF.BUFFER[in_Write_Index] := XUS_TN_SCREEN.bya_CHAR[in_Offset];

    				(* nächste Spalte anwählen *)
    				in_Offset := in_Offset + INT#01;
    			END_FOR

    			IF (bo_Break_Loop = TRUE) THEN;

    				(* Buffer Ende vorzeitig erreicht -> nur bis zur letzten kompletten Zeile uebertragen *)
    				in_Write_Index := in_Last_Row_Index;

    				EXIT;
    			END_IF

    			(* Buffer ist noch nicht voll -> neue Zeile ubernehmen *)
    			in_Last_Row_Index := in_Write_Index;
    			XUS_TN_SCREEN.bya_Line_Update[in_Row_Count] := FALSE;

    		END_IF

    		(* naechste Zeile adressieren *)
    		in_Row_Count := in_Row_Count + INT#01;

    		(* ab letzter Zeile wieder von vorne beginnen *)
    		IF (in_Row_Count > INT#23) THEN
    			in_Row_Count := INT#00;
    		END_IF
    		(*-----------------------------------------------*)

    	END_FOR

    	(* wenn in einen Update-Zyklus alle Zeilen auf einmal geschafft wurden *)
    	(* wird der Row_Count auf ersten Zeile gestellt *)
    	(* soll das hässliche Grafikflackern verhindern *)
    	(* ansonsten wird bei der letzen Zeile weitergemacht *)
    	IF (bo_Break_Loop = FALSE) THEN
    		in_Row_Count := INT#00;
    	END_IF

    	(* Edit-Cursor positionieren *)
    	IF (in_Write_Index <> in_Write_Index_Backup) THEN

    		in_Write_Index := in_Write_Index + INT#1;
    		S_BUF.BUFFER[in_Write_Index] := BYTE#16#1B; (* ESC *)
    		in_Write_Index := in_Write_Index + INT#1;
    		S_BUF.BUFFER[in_Write_Index] := BYTE#16#5B; (* [ *)

    		(* Zehnerstelle Zeilennummer ausgeben *)
    		in_Write_Index := in_Write_Index + INT#1;
    		S_BUF.BUFFER[in_Write_Index] := SHR(INT_TO_BCDC(XUS_TN_SCREEN.in_Cursor_Y + 1),INT#4) OR BYTE#16#30;

    		(* Einerstelle Zeilennummer ausgeben *)
    		in_Write_Index := in_Write_Index + INT#1;
    		S_BUF.BUFFER[in_Write_Index] := (INT_TO_BCDC(XUS_TN_SCREEN.in_Cursor_Y + 1) AND BYTE#16#0F) OR BYTE#16#30;

    		in_Write_Index := in_Write_Index + INT#1;
    		S_BUF.BUFFER[in_Write_Index] := BYTE#16#3B; (* ; *)

    		(* Zehnerstelle Spaltenummer ausgeben *)
    		in_Write_Index := in_Write_Index + INT#1;
    		S_BUF.BUFFER[in_Write_Index] := SHR(INT_TO_BCDC(XUS_TN_SCREEN.in_Cursor_X + 1),INT#4) OR BYTE#16#30;

    		(* Einerstelle Spaltennummer ausgeben *)
    		in_Write_Index := in_Write_Index + INT#1;
    		S_BUF.BUFFER[in_Write_Index] := (INT_TO_BCDC(XUS_TN_SCREEN.in_Cursor_X + 1) AND BYTE#16#0F) OR BYTE#16#30;

    		in_Write_Index := in_Write_Index + INT#1;
    		S_BUF.BUFFER[in_Write_Index] := BYTE#16#48; (* H *)

    END_IF

    (* aktuellen Schreibindex speichern -> Senden anstossen *)
    S_BUF.SIZE := INT_TO_UINT(in_Write_Index + 1);

    (* revision history
    ks	10. mai. 2010	rev 1.0
    	original version
    *)
END_FUNCTION_BLOCK

(* ---- UNI_CIRCULAR_BUFFER.st ---- *)
FUNCTION_BLOCK UNI_CIRCULAR_BUFFER
    (*http://www.oscat.de/images/OSCATNetwork/oscat_netlib121_en.pdf#page=69*)
    CASE DATA.D_MODE OF

    01:	x := WORD_TO_BYTE(DATA.D_HEAD); (* nur rechtes byte auswerten *)
    	CASE x OF
    	01:	cnt := LEN(DATA.D_STRING); (* String verarbeiten *)
    		pTmp := ADR(DATA.D_STRING);
    	02:	cnt := 4; (* Real verarbeiten *)
    		pTmp := ADR(DATA.D_REAL);
    	03:	cnt := 4; (* DWORD verarbeiten *)
    		pTmp := ADR(DATA.D_DWORD);
    	ELSE
    		cnt := 0;
    	END_CASE

    	DATA.BUF_DATA_CNT := DATA.BUF_DATA_CNT + UDINT#1;

    	(* ------ Daten in buffer eintragen ------ *)
    	buf_totalsize := SIZEOF(DATA.BUF);

    	IF (cnt + HeaderSize) > (buf_totalsize - DATA.BUF_SIZE) THEN (* genug Speicher frei ? *)
    		DATA.BUF_DATA_LOST := DATA.BUF_DATA_LOST + UDINT#1;
    		RETURN;
    	END_IF

    	DATA.D_SIZE := cnt;

    	mode_last := DATA.D_MODE;
    	tmp_dw := SHL(WORD_TO_DWORD(DATA.D_HEAD),16) OR UINT_TO_DWORD(cnt);

    	(* Header in Buffer eintragen *)
    	n1 := 0;
    	REPEAT
    		n2 := MIN(HeaderSize - n1, buf_totalsize - DATA._Last);
    		FOR n := 1 TO n2 DO
    			tmp_dw := ROL(tmp_dw,8);
    			DATA.BUF[DATA._Last] := DWORD_TO_BYTE(tmp_dw);
    			DATA._Last := DATA._Last + 1;
    		END_FOR
    		IF DATA._Last >= buf_totalsize THEN
    			DATA._Last := 0;
    		END_IF
    		n1 := n1 + n2;
    	UNTIL n1 >= HeaderSize
    	END_REPEAT

    	(* Daten in Buffer eintragen *)
    	n1 := 0;
    	REPEAT
    		n2 := MIN(cnt - n1, buf_totalsize - DATA._Last);
    		FOR n := 1 TO n2 DO
    			DATA.BUF[DATA._Last] := pTmp;
    			pTmp := pTmp + 1;
    			DATA._Last := DATA._Last + 1;
    		END_FOR
    		IF DATA._Last >= buf_totalsize THEN
    			DATA._Last := 0;
    		END_IF
    		n1 := n1 + n2;
    	UNTIL n1 >= cnt
    	END_REPEAT

    	DATA.BUF_SIZE := DATA.BUF_SIZE + cnt + HeaderSize;
    	DATA.BUF_COUNT := DATA.BUF_COUNT + 1;
    	DATA.BUF_USED := UINT_TO_USINT(100 * DATA.BUF_SIZE / buf_totalsize); (* benützer Speicher in % *)
    	DATA.D_MODE := 0;

    	(*####################  DEBUG-MESSAGE  ###################################*)
    	(*IF _debug_enable THEN
    		LOG_CL.NEW_MSG := 'RP: ADD /HEAD ~1 / SIZE ~2 / cnt ~3 / >~4<';
    		LOG_CL.PRINTF[1] := DWORD_TO_STRH(DATA.D_HEAD);
    		LOG_CL.PRINTF[2] := UINT_TO_STRING(cnt);
    		LOG_CL.PRINTF[3] := UINT_TO_STRING(DATA.BUF_COUNT);
    		CASE x OF
    		01:	LOG_CL.PRINTF[4] := DATA.D_STRING;
    		02:	LOG_CL.PRINTF[4] := REAL_TO_STRING(DATA.D_REAL);
    		03:	LOG_CL.PRINTF[4] := DWORD_TO_STRH(DATA.D_DWORD);
    		ELSE
    			LOG_CL.PRINTF[4] := '';
    		END_CASE
    		LOG_MSG();
    	END_IF*)
    	(*########################################################################*)

    10..12:	(* ------ Daten aus buffer auslesen und optional löschen ------ *)
    		(* 10 = nur lesen / 11 = löschen nach lesen / 12 = lesen und löschen *)
    	IF DATA.D_MODE <> 11 THEN
    		IF DATA.BUF_COUNT = 0 THEN RETURN; END_IF
    		buf_totalsize := SIZEOF(DATA.BUF);
    		DATA._GetEnd := DATA._First;(* index des ältesten eintrags merken *)
    		mode_last := DATA.D_MODE;

    		(* Header aus Buffer lesen *)
    		n1 := 0;
    		tmp_dw := 0;
    		REPEAT
    			n2 := MIN(HeaderSize - n1, buf_totalsize - DATA._GetEnd);
    			FOR n := 1 TO n2 DO
    				tmp_dw := ROL(tmp_dw,8) OR BYTE_TO_DWORD(DATA.BUF[DATA._GetEnd]);
    				DATA._GetEnd := DATA._GetEnd + 1;
    			END_FOR
    			IF DATA._GetEnd >= buf_totalsize THEN
    				DATA._GetEnd := 0;
    			END_IF
    			n1 := n1 + n2;
    		UNTIL n1 >= HeaderSize
    		END_REPEAT

    		DATA._GetStart := DATA._GetEnd;
    		cnt := DWORD_TO_UINT(tmp_dw AND 16#0000_FFFF);
    		DATA.D_SIZE := cnt;
    		DATA.D_HEAD := DWORD_TO_WORD(SHR(tmp_dw,16));

    		x := WORD_TO_BYTE(DATA.D_HEAD); (* nur rechtes byte auswerten *)
    		CASE x OF
    		01:	pTmp := ADR(DATA.D_STRING); (* String verarbeiten *)
    		02:	pTmp := ADR(DATA.D_REAL); (* Real verarbeiten *)
    		03:	pTmp := ADR(DATA.D_DWORD); (* DWORD verarbeiten *)
    		END_CASE

    		(* Daten aus Buffer lesen *)
    		n1 := 0;
    		REPEAT
    			n2 := MIN(cnt - n1, buf_totalsize - DATA._GetEnd);
    			FOR n := 1 TO n2 DO
    				pTmp := DATA.BUF[DATA._GetEnd];
    				pTmp := pTmp + 1;
    				DATA._GetEnd := DATA._GetEnd + 1;
    			END_FOR
    			IF DATA._GetEnd >= buf_totalsize THEN
    				DATA._GetEnd := 0;
    			END_IF
    			n1 := n1 + n2;
    		UNTIL n1 >= cnt
    		END_REPEAT
    		IF x = 1 THEN
    			pTmp := 0; (* String terminieren *)
    		END_IF
    		DATA.D_MODE := 0;

    		(*####################  DEBUG-MESSAGE  ###################################*)
    		(*IF _debug_enable THEN
    			LOG_CL.NEW_MSG := 'RP: READ /HEAD ~1 / SIZE ~2 / cnt ~3 / >~4<';
    			LOG_CL.PRINTF[1] := DWORD_TO_STRH(DATA.D_HEAD);
    			LOG_CL.PRINTF[2] := UINT_TO_STRING(cnt);
    			LOG_CL.PRINTF[3] := UINT_TO_STRING(DATA.BUF_COUNT);
    			CASE x OF
    			01:	LOG_CL.PRINTF[4] := DATA.D_STRING;
    			02:	LOG_CL.PRINTF[4] := REAL_TO_STRING(DATA.D_REAL);
    			03:	LOG_CL.PRINTF[4] := DWORD_TO_STRH(DATA.D_DWORD);
    			ELSE
    				LOG_CL.PRINTF[4] := '';
    			END_CASE
    			LOG_MSG();
    		END_IF*)
    		(*########################################################################*)
    	END_IF

    	IF (mode_last = 10 AND DATA.D_MODE = 11) OR (mode_last = 12 AND DATA.D_MODE = 0) THEN (* löschen nur direkt nach lesen möglich *)
    		mode_last := DATA.D_MODE;
    		DATA.BUF_SIZE := DATA.BUF_SIZE - cnt - HeaderSize;
    		DATA.BUF_COUNT := DATA.BUF_COUNT - 1;
    		DATA._First := DATA._GetEnd;
    		DATA.BUF_USED := UINT_TO_USINT(100 * DATA.BUF_SIZE / SIZEOF(DATA.BUF)); (* benützer Speicher in % *)
    		DATA.D_MODE := 0;

    		(*####################  DEBUG-MESSAGE  ###################################*)
    		(*IF _debug_enable THEN
    			LOG_CL.NEW_MSG := 'RP: DEL /HEAD ~1 / SIZE ~2 / cnt ~3 / >~4<';
    			LOG_CL.PRINTF[1] := DWORD_TO_STRH(DATA.D_HEAD);
    			LOG_CL.PRINTF[2] := UINT_TO_STRING(cnt);
    			LOG_CL.PRINTF[3] := UINT_TO_STRING(DATA.BUF_COUNT);
    			CASE x OF
    			01:	LOG_CL.PRINTF[4] := DATA.D_STRING;
    			02:	LOG_CL.PRINTF[4] := REAL_TO_STRING(DATA.D_REAL);
    			03:	LOG_CL.PRINTF[4] := DWORD_TO_STRH(DATA.D_DWORD);
    			ELSE
    				LOG_CL.PRINTF[4] := '';
    			END_CASE
    			LOG_MSG();
    		END_IF*)
    		(*########################################################################*)
    	END_IF

    99:	(* Buffer reset - alles löschen *)
    	DATA._First := 0;
    	DATA._Last := 0;
    	DATA._GetStart := 0;
    	DATA._GetEnd := 0;
    	DATA.BUF_COUNT := 0;
    	DATA.BUF_SIZE := 0;
    	DATA.BUF_USED := 0;
    	DATA.D_STRING := '';
    	DATA.D_DWORD := 0;
    	DATA.D_REAL := 0.0;
    	DATA.D_HEAD := 0;
    	DATA.D_MODE := 0;
    	DATA.D_SIZE := 0;
    	mode_last := 0;
    END_CASE

    (* höchsten Auslastungswert speichern *)
    IF DATA.BUF_USED > DATA.BUF_USED_MAX THEN
    	DATA.BUF_USED_MAX := DATA.BUF_USED;
    END_IF

    (* revision history
    ks	01. jan. 2011	rev 1.0
    	original version
    ks	25. jul. 2011	rev 1.1
    	neuen MODE 12 hinzugefügt
    ks	03. Sep. 2015	rev 1.2
    	Auslastungsüberwachung hinzugefügt
    ks	21. mar. 2016	rev 1.3
    	D_SIZE info hinzugefügt
    	Buffer size auf 8192 vergroessert
    *)
END_FUNCTION_BLOCK

(* ---- WORLD_WEATHER.st ---- *)
FUNCTION_BLOCK WORLD_WEATHER
    (*http://www.oscat.de/images/OSCATNetwork/oscat_netlib121_en.pdf#page=211*)
    CASE state OF

    00:
    	IF ACTIVATE AND NOT last_state THEN
    		state := 20;
    		DONE := FALSE;
    		BUSY := TRUE;
    		ERROR_C := DWORD#0;
    		ERROR_T := BYTE#0;
    	END_IF

    20: (* URL for DNS UND HTTP-GET *)
    	(* Example: http://api.worldweatheronline.com/free/v1/weather.ashx?q=48.21,16.37&format=csv&num_of_days=5&KEY=xxxxxxxxxxxxxxxxxxxxxx *)
    	url_str := CONCAT('http://api.worldweatheronline.com/free/v1/weather.ashx?q=',REAL_TO_STRF(LATITUDE,6,D:='.'));
    	url_str := CONCAT(url_str,',');
    	url_str := CONCAT(url_str,REAL_TO_STRF(LONGITUDE,6,D:='.'));
    	url_str := CONCAT(url_str,'&format=csv&num_of_days=5&KEY=');
    	url_str := CONCAT(url_str,KEY);

    	URL_DATA:=STRING_TO_URL(STR:=url_str, DEFAULT_PROTOCOL:='', DEFAULT_PATH:='' );
    	state := 40;

    40:
    	IF DNS_CLIENT.DONE THEN
    		state := 60;
    	ELSIF (DNS_CLIENT.ERROR > DWORD#00) THEN
    		(* Fehlerbehandlung *)
    		ERROR_C := DNS_CLIENT.ERROR;
    	ERROR_T := BYTE#01;
    		state   := 100;
    	END_IF

    60:
    	IF HTTP_GET.DONE THEN
    		sep := 0;
    		idx := 0;
    		day := 0;
    		cnt := 0;
    		offset := HTTP_GET.BODY_START; (* Start offset vorgeben *)
    		size := HTTP_GET.BODY_STOP; (* End Position *)
    		run := 1; (* Element suchen *)
    		state := 80;

    	ELSIF (HTTP_GET.ERROR > DWORD#00) THEN
    		(* Fehlerbehandlung *)
    		ERROR_C := HTTP_GET.ERROR;
    		ERROR_T := BYTE#02;
    		state := 100;
    	END_IF

    80:	IF run = 0 THEN (* kein Befehl mehr aktiv ? *)
    		run := 1; (*  nächstes Element suchen  *)
    		IF result = 1 OR result = 2 THEN
    			value_int := 0;
    			value_real := 0.0;
    			(* automatische konvertierung in real und int ausführen *)
    			IF LEN(value) <= 20 THEN
    				v_real:=FLOAT_TO_REAL(FLT:=value);
    				IF CHK_REAL(v_real) = 0 THEN (* !!! prüft auf gültigen REAL Wert, ansonsten stürzt Twincat ab !!!!  *)
    					value_real := v_real;
    					value_int := REAL_TO_INT(value_real);
    				END_IF
    			END_IF
    			cnt := cnt + 1;

    			IF cnt = 1 AND LEFT(value,1) <> '#' THEN
    				cnt := 0;
    			END_IF

    			IF cnt >=8 AND cnt <= 87 THEN
    				IF cnt > 22 THEN
    					CASE idx OF
    					00:	WW.day[day].DATE_OF_DAY := value;
    					01:	WW.day[day].TEMP_MAX_C := value_int;
    					02:	WW.day[day].TEMP_MAX_F := value_int;
    					03:	WW.day[day].TEMP_MIN_C := value_int;
    					04:	WW.day[day].TEMP_MIN_F := value_int;
    					05:	WW.day[day].WIND_SPEED_MILES := value_int;
    					06:	WW.day[day].WIND_SPEED_KMPH := value_int;
    					07:	WW.day[day].WIND_DIR_DEGREE := value_int;
    					08:	WW.day[day].WIND_DIR16POINT := value;
    					09:	WW.day[day].WEATHER_CODE := value_int;
    					10:	pos := FIND(value, '/wsymbol_');
    						WW.day[day].WEATHER_ICON := DEC_TO_INT(MID(value,4,pos+9));
    					11:	WW.day[day].WEATHER_DESC := value;
    					12:	WW.day[day].PRECIPMM := value_real;
    					END_CASE
    					idx := idx + 1;
    					IF idx > 12 THEN
    						idx := 0;
    						day := day + 1;
    					END_IF
    				ELSE
    					CASE cnt OF
    					08:	sep :=44; (* ab jetzt mit Trennzeichen arbeiten, *)
    					09:	WW.CUR.OBSERVATION_TIME := value;
    					10:	WW.CUR.TEMP_C := value_int;
    					11:	WW.CUR.WEATHER_CODE := value_int;
    					12:	pos := FIND(value, '/wsymbol_');
    						WW.CUR.WEATHER_ICON := DEC_TO_INT(MID(value,4,pos+9));
    					13:	WW.CUR.WEATHER_DESC := value;
    					14:	WW.CUR.WIND_SPEED_MILES := value_int;
    					15:	WW.CUR.WIND_SPEED_KMPH := value_int;
    					16:	WW.CUR.WIND_DIR_DEGREE := value_int;
    					17:	WW.CUR.WIND_DIR16POINT := value;
    					18:	WW.CUR.PRECIPMM := value_real;
    					19:	WW.CUR.HUMIDITY := value_int;
    					20:	WW.CUR.VISIBILITY := value_int;
    					21:	WW.CUR.PRESSURE := value_int;
    					22:	WW.CUR.CLOUDOVER := value_int;
    					END_CASE
    				END_IF
    			END_IF
    		ELSIF result = 10 THEN (* nichts mehr gefunden *)
    			DONE  := TRUE;
    			run := 0; (* Auswertung beenden *)
    			state := 100;
    		END_IF
    	END_IF

    100:
    	(* UNLOCK HTTP DATA *)
    	IF (NOT HTTP_GET.DONE) THEN
    		state := 0;
    		BUSY := FALSE;
    		DONE := ERROR_T = BYTE#0;
    	END_IF

    END_CASE

    (* ---------------- DNS --------------- *)
    DNS_CLIENT(	IP_C:=IP_C,
    			S_BUF:=S_BUF,
    			R_BUF:=R_BUF,
    			DOMAIN:=URL_DATA.DOMAIN,
    			IP4_DNS:=DWORD#00,
    			ACTIVATE:=state=40 (* DNS Start *)
    			);
    (* nicht oder nicht direkt verwendete Parameter *)
    (*	DWORD :=DNS_CLIENT.IP4;
    	BOOL  :=DNS_CLIENT.DONE;
    	BYTE  :=DNS_CLIENT.ERROR; *)
    (* -------------------------------------*)

    (* ------------- HTTP_GET --------------- *)
    HTTP_GET(	IP_C:=IP_C,
    			S_BUF:=S_BUF,
    			R_BUF:=R_BUF,
    			IP4:=DNS_CLIENT.IP4,
    			GET:=state=60,
    			MODE:=BYTE#2, (* HTTP 1.1 mit persistenter Verbindung *)
    			UNLOCK_BUF:=state=100,
    			URL_DATA:=URL_DATA
    			);

    (* nicht oder nicht direkt verwendete Parameter *)
    (*	STRING := HTTP_GET.HTTP_STATUS;
    	UINT :=HTTP_GET.HEADER_START;
    	UINT :=HTTP_GET.HEADER_STOP;
    	UINT :=HTTP_GET.BODY_START;
    	UINT :=HTTP_GET.BODY_STOP;
    	BOOL :=HTTP_GET.DONE;
    	BYTE :=HTTP_GET.ERROR;
    *)
    (* -------------------------------------*)
    CPB(sep:=sep,run:=run,offset:=offset,value:=value,PT:=R_BUF,result=>result); (* CSV PARAMETER BUF *)

    last_state := ACTIVATE;

    (* revision history
    ks	01.oct. 2010	rev 1.0
    	original version

    ks	01.feb. 2011	rev 1.1
    	rücksetzen von cnt

    ks	07.apr. 2011	rev 1.2
    	neue Domain "free.worldweatheronline.com" (Ab 30.04.2011 notwendig)

    ks	05.jan. 2012	rev 1.3
    	neues datenelement "icon" integriert, REAL_TO_STRF parameter D

    ks	05.oct. 2012	rev 1.4
    	workaround für chunked html data

    ks	11.may. 2013	rev 1.5
    	New worldwaether url and api KEY required (new API-Services)
    *)
END_FUNCTION_BLOCK

(* ---- WORLD_WEATHER_DESC_GE.st ---- *)
FUNCTION_BLOCK WORLD_WEATHER_DESC_GE
    (*http://www.oscat.de/images/OSCATBasic/oscat_basic333_en.pdf#page=210*)
    IF ACTIVATE AND act_last = FALSE THEN
    	i := 0;
    	FOR y := 1 TO 12 DO
    		CASE y OF
    		1,3,5,7,9:		x :=  WW.DAY[i].WEATHER_CODE;
    		2,4,6,8,10:	WW.DAY[i].WEATHER_DESC := str;
    					i := i + 1;
    		11:			x :=  WW.CUR.WEATHER_CODE;
    		12:			WW.CUR.WEATHER_DESC := str;
    		END_CASE

    		CASE x OF
    			113	:	str := 'heiter/sonnig';
    			116	:	str := 'stellenweise wolkig';
    			119	:	str := 'wolkig';
    			122	:	str := 'bewölkt';
    			143	:	str := 'Nebel';
    			176	:	str := 'stellenweise nahegelegener Regen';
    			179	:	str := 'stellenweise nahegelegener Schneefall';
    			182	:	str := 'stellenweise nahegelegener Eisregen';
    			185	:	str := 'stellenweise gefrierender Niesel';
    			200	:	str := 'nahegelegene Sturm';
    			227	:	str := 'Schneetreiben';
    			230	:	str := 'Schneesturm';
    			248	:	str := 'Nebel';
    			260	:	str := 'gefrierender Nebel';
    			263	:	str := 'stellenweise leichter Nieselregen';
    			266	:	str := 'leichter Niesel';
    			281	:	str := 'gefrierender Nieselregen';
    			284	:	str := 'stark gefrierender Nieselregen';
    			293	:	str := 'stellenweise leichter Regen';
    			296	:	str := 'leichter Regen';
    			299	:	str := 'zeitweise etwas Regen';
    			302	:	str := 'mäßiger Regen';
    			305	:	str := 'zeitweise etwas starker Regen';
    			308	:	str := 'starker Regen';
    			311	:	str := 'leichter gefrierender Regen';
    			314	:	str := 'mäßiger oder starker Eisregen';
    			317	:	str := 'leichter Eisregen';
    			320	:	str := 'mäßiger oder starker Eisregen';
    			323	:	str := 'stellenweise leichter Schneefall';
    			326	:	str := 'leichter Scheefall';
    			329	:	str := 'stellenweise moderater Schneefall';
    			332	:	str := 'mäßiger Schnee';
    			335	:	str := 'stellenweise starker Scheefall';
    			338	:	str := 'starker Schneefall';
    			350	:	str := 'Hagel';
    			353	:	str := 'leichte Regenfälle';
    			356	:	str := 'mäßiger oder starker Regenfall';
    			359	:	str := 'sintflutartige Regenfälle';
    			362	:	str := 'leichter Eisregen';
    			365	:	str := 'mäßiger oder starker Eisregen';
    			368	:	str := 'leichte Schneeschauer';
    			371	:	str := 'mäßiger oder starker Schneefall';
    			374	:	str := 'leichter Hagel';
    			377	:	str := 'mäßiger oder starker Hagel';
    			386	:	str := 'stellenweise leichter Regen in Gewittergebiet';
    			389	:	str := 'mäßiger oder starker Regen in Gewittergebiet';
    			392	:	str := 'stellenweise leichter Schneefall in Gewittergebiet';
    			395	:	str := 'mäßiger oder starker Schnee in Gewittergebiet';
    		ELSE
    			str := 	'nicht verfügbar';
    		END_CASE
    	END_FOR
    END_IF
    act_last := ACTIVATE;

    (* revision history
    ks	04. may. 2011	rev 1.0
    	original version
    *)
END_FUNCTION_BLOCK

(* ---- WORLD_WEATHER_ICON_OSCAT.st ---- *)
FUNCTION_BLOCK WORLD_WEATHER_ICON_OSCAT
    (*http://www.oscat.de/images/OSCATNetwork/oscat_netlib121_en.pdf#page=215*)
    IF ACTIVATE AND act_last = FALSE THEN
    	x := LIMIT(0,WW.CUR.WEATHER_ICON,41);
    	WW.CUR.WEATHER_ICON := dat[x];
    	FOR i := 0 TO 4 DO
    		x := LIMIT(0,WW.DAY[i].WEATHER_ICON,41);
    		WW.DAY[i].WEATHER_ICON := dat[x];
    	END_FOR
    END_IF
    act_last := ACTIVATE;

    (* revision history
    ks	04. may. 2011	rev 1.0
    	original version
    *)
END_FUNCTION_BLOCK

(* ---- XML_READER.st ---- *)
FUNCTION_BLOCK XML_READER
    (*http://www.oscat.de/images/OSCATNetwork/oscat_netlib121_en.pdf#page=140*)
    (*

    TYP
    00 = UNBEKANNT
    01 = ELEMENT (STANDARD)
    02 = CLOSE ELEMENT
    03 = TEXT
    04 = ATTRIBUTE
    05 = ELEMENT (PROCESSING INSTRUCTION)

    12 = !CDATA
    13 = !COMMENT
    14 = !DTD ELEMENT (Document Type Declarations )

    98 = watchdog
    99 = ENDE

    Bei Typ 02 werden keine Blockdaten ausgegeben !

    *)

    (* ---------- Init -------------- *)
    IF BIT_OF_DWORD(WORD_TO_DWORD(CTRL.command),15) THEN
    	command := CTRL.command;
    	CTRL.command := WORD#0;

    	index := UINT_TO_INT(CTRL.START_POS);
    	stop := UINT_TO_INT(CTRL.STOP_POS);
    	mode := 100;
    	path_overflow := FALSE;

    	CTRL.TYP := 0;
    	CTRL.COUNT := UINT#00;
    	CTRL.LEVEL := UINT#00;
    	CTRL.ATTRIBUTE := '';
    	CTRL.ELEMENT := '';
    	CTRL.PATH := '';
    	CTRL.VALUE := '';

    	watchdog.PT := CTRL.watchdog;
    END_IF

    (*----------------------------------------------- *)

    IF index < 0 THEN RETURN;END_IF

    CTRL.BLOCK1_START := UINT#0;
    CTRL.BLOCK1_STOP := UINT#0;
    CTRL.BLOCK2_START := UINT#0;
    CTRL.BLOCK2_STOP := UINT#0;

    watchdog(IN:=FALSE); (* Timer stoppen *)

    WHILE (TRUE) DO

    	(* -------------- watchdog ------------------ *)
    	watchdog(IN:=CTRL.watchdog > T#0s);
    	IF watchdog.Q THEN
    		CTRL.TYP := 98;
        		(*####################  DEBUG-MESSAGE  ###################################*)
        		(*IF _debug_enable THEN
          			LOG_CL.NEW_MSG := 'watchdog:';
          			LOG_MSG();
        		END_IF*)
        		(*########################################################################*)
    		RETURN;
    	END_IF

    	(* -------------- PARSING END ------------------ *)
    	IF index > stop THEN
    		CTRL.COUNT := CTRL.COUNT + UINT#1;
    		CTRL.TYP := 99;
        		(*####################  DEBUG-MESSAGE  ###################################*)
        		(*IF _debug_enable THEN
          			LOG_CL.NEW_MSG := 'EX: #T:~1 #c:~2 #P:~6 #L:~7';
          			LOG_CL.PRINTF[1] := INT_TO_STRING(CTRL.TYP);
          			LOG_CL.PRINTF[2] := UINT_TO_STRING(CTRL.COUNT);
          			LOG_CL.PRINTF[6] := CTRL.PATH;
          			LOG_CL.PRINTF[7] := UINT_TO_STRING(CTRL.LEVEL);
          			LOG_MSG();
        		END_IF*)
        		(*########################################################################*)
    		mode  := 0; (* Schritt ruecksetzen *)
    		index := 0; (* Abarbeitung stoppen *)
    		RETURN;
    	END_IF

    	CASE mode OF

    	100: (* ---------- ELEMENT SECTION ------------------ *)
    		(* search begin of element *)
    		s1 := 0;
    		e1 := 0;
    		WHILE (index <= stop) DO
    			IF BUF[index]=BYTE#60 THEN (* '<' TagBegin *)
    				index := index + 1;
    				c := BUF[index];
    				IF c = BYTE#47 THEN (* '/' TagTerm *)
    					mode := 300; (* End Element Section *)
    				ELSIF c = BYTE#33 THEN (* '!' for Special Section *)
    					index := index + 1;
    					mode := 500;
    				ELSE
    					s1 := index;
    				END_IF
    				EXIT;
    			END_IF
    			index := index + 1;
    		END_WHILE

    		(* analyse element *)
    		CTRL.TYP := 0; (* TYP löschen *)
    		IF s1 > 0 THEN
    			WHILE (index <= stop AND e1 = 0) DO
    				c := BUF[index];
    				(* whitespace zeichen = Element with Attributes *)
    				IF c <= BYTE#32 THEN
    					(* suche nächstes druckbares zeichen *)
    					index2 := index;
    					WHILE (index2 <= stop) AND (BUF[index2] <= BYTE#32) DO
    						index2 := index2 + 1;
    					END_WHILE
    					IF BUF[index2] = BYTE#47 THEN (* pruefe auf leeres Element '/' *)
    						index := index2;
    						e1 := index - 2;
    						CTRL.TYP := 1; (* struktur-element *)
    						mode := 300;   (* Close Element *)
    						EXIT;
    					END_IF

    					e1 := index - 1;
    					CTRL.TYP := 1; (* Element mit Attribute *)
    					mode := 400;

    				ELSIF c = BYTE#62 THEN (* '>' TagEnd *)

    					(* pruefe auf leeres Element <xx/> *)
    					index2 := index - 1;
    					IF BUF[index2] = BYTE#47 THEN (* TagTerm '/' *)
    						e1 := index2 - 1;
    						CTRL.TYP := 1;
    						empty_tag := TRUE; (* EMPTY TAG mode *)
    						mode := 200; (* TEXT Element *)
    						EXIT;
    					END_IF

    					e1 := index - 1;
    					index2 := index + 1;

    					(* untersuche nachfolgendes Element *)
    					WHILE (index2 <= stop) DO
    						c := BUF[index2];
    						IF c = BYTE#60 THEN (* '<' TagBegin *)

    							index2 := index2 + 1; (* geht bei PCWORX leider nicht anders !*)
    							c := BUF[index2];
    							index2 := index2 - 1;
    							IF c = BYTE#47 THEN (* TagTerm '/' *)
    								empty_tag := TRUE;
    								mode := 200; (* TEXT Element *)
    							ELSE
    								mode := 100; (* Element *)
    							END_IF
    							CTRL.TYP := 1; (* struktur-element *)
    							EXIT;
    						ELSIF c > BYTE#32  THEN (* Printable-Character *)
    							CTRL.TYP := 1; (* element with text *)
    							mode := 200;
    							EXIT;
    						END_IF
    						index2 := index2 + 1;
    					END_WHILE
    				END_IF
    				index := index + 1;
    			END_WHILE
    		END_IF

    		(* Neues Element gefunden*)
    		IF CTRL.TYP > 0 THEN

    			(* Sonderprüfung auf Processing Instruction (PI) *)
    			IF BUF[s1] = BYTE#63 THEN (* '?' for Processing Instruction *)
    				s1 := s1 + 1; (* führendes '?' auslassen *)
    				CTRL.TYP := 5;
    			END_IF
    			CTRL.BLOCK1_START := INT_TO_UINT(s1);
    			CTRL.BLOCK1_STOP  := INT_TO_UINT(e1);
    			CTRL.ELEMENT := BUFFER_TO_STRING(PT:=ADR(BUF),SIZE:=INT_TO_UINT(stop + 1),START:=CTRL.BLOCK1_START,stop:=CTRL.BLOCK1_STOP);
    			CTRL.COUNT := CTRL.COUNT + UINT#1;
    			CTRL.LEVEL := CTRL.LEVEL + UINT#1;

    			IF path_overflow = FALSE THEN
    				(* Stringlänge überwachen *)
    				IF LEN(CTRL.PATH) + LEN(CTRL.ELEMENT) + 1 > 250 THEN
    					path_overflow := TRUE;
    					CTRL.PATH := 'OVERFLOW';
    				ELSE
    					CTRL.PATH := CONCAT(CTRL.PATH,'/');
    					CTRL.PATH  := CONCAT(CTRL.PATH,CTRL.ELEMENT);
    				END_IF
    			END_IF

    			IF BIT_OF_DWORD(WORD_TO_DWORD(command),CTRL.TYP) THEN
            				(*####################  DEBUG-MESSAGE  ###################################*)
            				(*IF _debug_enable THEN
              				LOG_CL.NEW_MSG := 'EL: #T:~1 #c:~2 #E:~3 #P:~6 #L:~7';
              				LOG_CL.PRINTF[1] := INT_TO_STRING(CTRL.TYP);
              				LOG_CL.PRINTF[2] := UINT_TO_STRING(CTRL.COUNT);
              				LOG_CL.PRINTF[3] := CTRL.ELEMENT;
              				LOG_CL.PRINTF[6] := CTRL.PATH;
              				LOG_CL.PRINTF[7] := UINT_TO_STRING(CTRL.LEVEL);
              				LOG_MSG();
            				END_IF*)
            				(*########################################################################*)
    				RETURN;
    			END_IF
    		END_IF

    	200: (* ---------- TEXT SECTION ------------------ *)
    		CTRL.VALUE := '';
    		IF empty_tag = FALSE THEN
    			s1 := index;
    			(* suche '<' EndTag*)
    			WHILE (index <= stop) AND (BUF[index] <> BYTE#60) DO
    				index := index + 1;
    			END_WHILE

    			e1 := index - 1;
    			CTRL.BLOCK1_START := INT_TO_UINT(s1);
    			CTRL.BLOCK1_STOP  := INT_TO_UINT(e1);
    			CTRL.VALUE := BUFFER_TO_STRING(PT:=ADR(BUF),SIZE:=INT_TO_UINT(stop + 1),START:=CTRL.BLOCK1_START,stop:=CTRL.BLOCK1_STOP);
    		END_IF

    		empty_tag := FALSE;
    		mode := 300; (* -> NEXT-JOB: END ELEMENT *)
    		CTRL.COUNT := CTRL.COUNT + UINT#1;
    		CTRL.TYP := 3;

    		IF BIT_OF_DWORD(WORD_TO_DWORD(command),CTRL.TYP) THEN
          			(*####################  DEBUG-MESSAGE  ###################################*)
          			(*IF _debug_enable THEN
            				LOG_CL.NEW_MSG := 'TE: #T:~1 #c:~2 #E:~3 #V:~4 #P:~6 #L:~7';
            				LOG_CL.PRINTF[1] := INT_TO_STRING(CTRL.TYP);
            				LOG_CL.PRINTF[2] := UINT_TO_STRING(CTRL.COUNT);
            				LOG_CL.PRINTF[3] := CTRL.ELEMENT;
            				LOG_CL.PRINTF[4] := CTRL.VALUE;
            				LOG_CL.PRINTF[6] := CTRL.PATH;
            				LOG_CL.PRINTF[7] := UINT_TO_STRING(CTRL.LEVEL);
            				LOG_MSG();
          			END_IF*)
          			(*########################################################################*)
    			RETURN;
    		END_IF

    	300: (* ---------- END ELEMENT SECTION ------------------ *)
    		WHILE (index <= stop) DO
    			c := BUF[index];
    			IF c = BYTE#62 THEN (* '>' TagEnd *)
    				index := index + 1;
    				s1 := FINDB(str1:=CTRL.PATH,str2:='/');
    				IF path_overflow = FALSE THEN
    					IF s1 > 1 THEN
    						CTRL.ELEMENT := RIGHT(CTRL.PATH,LEN(CTRL.PATH) - s1);
    						CTRL.PATH := LEFT(CTRL.PATH,s1 - 1);
    					ELSE
    						CTRL.ELEMENT := RIGHT(CTRL.PATH,LEN(CTRL.PATH) - 1);
    						CTRL.PATH :='';
    					END_IF
    				END_IF

    				CTRL.LEVEL := CTRL.LEVEL - UINT#1;
    				CTRL.COUNT := CTRL.COUNT + UINT#1;
    				CTRL.TYP := 2;
    				mode := 100;

    				IF BIT_OF_DWORD(WORD_TO_DWORD(command),CTRL.TYP) THEN
             	 				(*####################  DEBUG-MESSAGE  ###################################*)
              				(*IF _debug_enable THEN
                					LOG_CL.NEW_MSG := 'CE: #T:~1 #c:~2 #E:~3 #P:~6 #L:~7';
                					LOG_CL.PRINTF[1] := INT_TO_STRING(CTRL.TYP);
                					LOG_CL.PRINTF[2] := UINT_TO_STRING(CTRL.COUNT);
                					LOG_CL.PRINTF[3] := CTRL.ELEMENT;
                					LOG_CL.PRINTF[6] := CTRL.PATH;
                					LOG_CL.PRINTF[7] := UINT_TO_STRING(CTRL.LEVEL);
                					LOG_MSG();
              				END_IF*)
              				(*########################################################################*)
    					RETURN;
    				ELSE
    					EXIT;
    				END_IF
    			END_IF
    			index := index + 1;
    		END_WHILE

    	400: (* ---------- ATTRIBUTE SECTION ------------------ *)
    		(* search first normal charakter *)
    		WHILE (index <= stop AND BUF[index] <= BYTE#32) DO
    			index := index + 1;
    		END_WHILE

    		(* begin Attribe name *)
    		e1 := 0;
    		s1 := index;
    		(* search end of Attrib Name '=' *)
    		WHILE (index <= stop) DO
    			IF BUF[index] = BYTE#61 THEN (* '=' Equals *)
    				e1 := index - 1;
    				EXIT;
    			END_IF
    			index := index + 1;
    		END_WHILE

    		IF e1 > 0 THEN
    			(* Attribute Name *)
    			CTRL.BLOCK1_START := INT_TO_UINT(s1);
    			CTRL.BLOCK1_STOP  := INT_TO_UINT(e1);
    			CTRL.ATTRIBUTE := BUFFER_TO_STRING(PT:=ADR(BUF),SIZE:=INT_TO_UINT(stop + 1),START:=CTRL.BLOCK1_START,stop:=CTRL.BLOCK1_STOP);
    			(* search end of Attrib Value '=' *)
    			index := index + 2;
    			e1 := 0;
    			s1 := index;
    			WHILE (index <= stop AND e1 = 0) DO
    				c := BUF[index];
    				IF c = BYTE#34 OR c = BYTE#39 THEN (* " OR ' Equals *)
    					e1 := index - 1;
    				END_IF
    				index := index + 1;
    			END_WHILE

    			IF e1 > 0 THEN
    				(* Value *)
    				CTRL.BLOCK2_START := INT_TO_UINT(s1);
    				CTRL.BLOCK2_STOP  := INT_TO_UINT(e1);

    				(* bei leeren "" ist start groesser als stop und wird somit zum leerstring *)
    				CTRL.VALUE := BUFFER_TO_STRING(PT:=ADR(BUF),SIZE:=INT_TO_UINT(stop + 1),START:=CTRL.BLOCK2_START,stop:=CTRL.BLOCK2_STOP);
    				(* search next non white space charakter *)
    				WHILE (index <= stop AND BUF[index] <= BYTE#32) DO
    					index := index + 1;
    				END_WHILE

    					c := BUF[index];
    					(* TagEnd '>' *)
    					IF c = BYTE#62 THEN
    						index := index + 1;
    						index2 := index;

    					(* search next non white space charakter *)
    					WHILE (index <= stop AND BUF[index] <= BYTE#32) DO
    						index := index + 1;
    					END_WHILE

    					IF BUF[index] = BYTE#60 THEN (* TagBegin '<' *)
    						mode := 100; (* -> NEXT-JOB: ELEMENT-SECTION *)
    					ELSE
    						index := index2;
    						mode := 200; (* -> NEXT-JOB: TEXT-SECTION *)
    					END_IF

    				ELSIF c = BYTE#47 OR c = BYTE#63 THEN (* TagTerm '/' OR '?' end Processing Instruction *)
    					mode := 300; (* -> NEXT-JOB: END ELEMENT *)
    				ELSE
    					mode := 400; (* -> NEXT-JOB: ATTRIBUTE-SECTION *)
    				END_IF

    				CTRL.COUNT := CTRL.COUNT + UINT#1;
    				CTRL.TYP := 4;
    				IF BIT_OF_DWORD(WORD_TO_DWORD(command),CTRL.TYP) THEN
              				(*####################  DEBUG-MESSAGE  ###################################*)
              				(*IF _debug_enable THEN
                					LOG_CL.NEW_MSG := 'AT: #T:~1 #c:~2 #E:~3 #A:~4 #V:~5 #P:~6 #L:~7';
                					LOG_CL.PRINTF[1] := INT_TO_STRING(CTRL.TYP);
                					LOG_CL.PRINTF[2] := UINT_TO_STRING(CTRL.COUNT);
                					LOG_CL.PRINTF[3] := CTRL.ELEMENT;
                					LOG_CL.PRINTF[4] := CTRL.ATTRIBUTE;
                					LOG_CL.PRINTF[5] := CTRL.VALUE;
                					LOG_CL.PRINTF[6] := CTRL.PATH;
                					LOG_CL.PRINTF[7] := UINT_TO_STRING(CTRL.LEVEL);
                					LOG_MSG();
              				END_IF*)
              				(*########################################################################*)
    					RETURN;
    				END_IF
    			END_IF
    		END_IF

    	500: (* ---------- SPECIAL DATA SECTION (Document Type Declarations) ---------- *)

    		CTRL.TYP := 0;
    		s1 := 0;
    		index2 := 11;

    		WHILE (s1 = 0) DO
    			index2 := index2 + 1;
    			CTRL.TYP := index2;

    			CASE index2 OF
    			12: (* CDATA *)
    				s_code := '[CDATA[';
    				e_code := ']]>';
    			13: (* COMMENT *)
    				s_code := '--';
    				e_code := '-->';
    			14: (* ANY DTD *)
    				e_code := '';
    				s1 := index;
    				EXIT;
    			END_CASE

    			e1 := LEN(s_code);
    			IF BUFFER_SEARCH(PT:=ADR(BUF),SIZE:=INT_TO_UINT(index + e1),STR:=s_code,POS:=index,IGN:=FALSE) = index THEN
    				s1 := index + e1;
    			END_IF
    		END_WHILE

    		CTRL.BLOCK1_START := INT_TO_UINT(s1);
    		IF LEN(e_code) > 0 THEN
    			(* Ende Kennung suchen *)
    			e1 := BUFFER_SEARCH(PT:=ADR(BUF),SIZE:=INT_TO_UINT(stop + 1),STR:=e_code,POS:=index,IGN:=FALSE);
    			CTRL.BLOCK1_STOP := INT_TO_UINT(e1 - 1);
    			index := e1 + LEN(e_code); (* naechstes element *)
    		ELSE
    			(* suche '>' EndTag*)
    			index2 := 1; (* <> Paar zähler *)
    			WHILE (index <= stop AND index2 > 0) DO
    				c := BUF[index];
    				IF c = BYTE#60 THEN (* '<' TagBegin *)
    					index2 := index2 + 1;
    				ELSIF c = BYTE#62 THEN (* '>' TagEnd   *)
    					index2 := index2 - 1;
    				ELSIF c = BYTE#34 OR c = BYTE#39 THEN (* " Double Quote OR ' Single Quote *)
    					index := index + 1;
    					WHILE (index <= stop) DO
    						c := BUF[index];
    						IF c = BYTE#34 OR c = BYTE#39 THEN (* " Double Quote OR ' Single Quote *)
    							EXIT;
    						END_IF
    						index := index + 1;
    					END_WHILE
    				END_IF
    				index := index + 1;
    			END_WHILE
    			CTRL.BLOCK1_STOP := INT_TO_UINT(index - 2);
    		END_IF

    		CTRL.VALUE := BUFFER_TO_STRING(PT:=ADR(BUF),SIZE:=INT_TO_UINT(stop + 1),START:=CTRL.BLOCK1_START,stop:=CTRL.BLOCK1_STOP);
    		CTRL.COUNT := CTRL.COUNT + UINT#1;
    		mode := 100; (* -> NEXT-JOB: ELEMENT *)

    		IF BIT_OF_DWORD(WORD_TO_DWORD(command),CTRL.TYP) THEN
          			(*####################  DEBUG-MESSAGE  ###################################*)
          			(*IF _debug_enable THEN
            				LOG_CL.NEW_MSG := 'DTD: #T:~1 #c:~2 #S:~3 #E:~4 #V:~5 #P:~6 #L:~7';
            				LOG_CL.PRINTF[1] := INT_TO_STRING(CTRL.TYP);
            				LOG_CL.PRINTF[2] := UINT_TO_STRING(CTRL.COUNT);
            				LOG_CL.PRINTF[3] := UINT_TO_STRING(CTRL.BLOCK1_START);
            				LOG_CL.PRINTF[4] := UINT_TO_STRING(CTRL.BLOCK1_STOP);
            				LOG_CL.PRINTF[5] := CTRL.VALUE;
            				LOG_CL.PRINTF[6] := CTRL.PATH;
            				LOG_CL.PRINTF[7] := UINT_TO_STRING(CTRL.LEVEL);
            				LOG_MSG();
          			END_IF*)
          			(*########################################################################*)
    			RETURN;
    		END_IF

    	END_CASE
    END_WHILE

    (* revision history
    ks	18. oct. 2008	rev 1.0
    	original version

    ks	20. oct. 2009	rev 1.1
    	Networkbuffer und Buffer-funktionen auf Basis 0

    ks	10. mai. 2010	rev 1.2
    	stringlänge maximal 250 zeichen

    *)
END_FUNCTION_BLOCK

(* ---- YAHOO_WEATHER.st ---- *)
FUNCTION_BLOCK YAHOO_WEATHER
    (*http://www.oscat.de/images/OSCATNetwork/oscat_netlib121_en.pdf#page=207*)
    (* read system time *)
    tx := T_PLC_MS();

    CASE state OF

    00:	IF ACTIVATE AND NOT activate_last THEN
    		state := 40;
    		DONE := FALSE;
    		BUSY := TRUE;
    		ERROR_C := DWORD#0;
    		ERROR_T := BYTE#0;
    		cycle := 0;
    		repeat_count := USINT#0;
    		repeat_request := FALSE;
      		URL_DATA.DOMAIN := 'query.yahooapis.com'; (* Domainname für DNS_CLIENT *)
    	END_IF

    40:	IF DNS_CLIENT.DONE THEN
    		state := 50;
    	ELSIF (DNS_CLIENT.ERROR > DWORD#00) THEN
    		(* Fehlerbehandlung *)
    		ERROR_C := DNS_CLIENT.ERROR;
    		ERROR_T := BYTE#01;
    		state   := 100;
    	END_IF

    50:   	(* Teil 1: http://query.yahooapis.com/v1/public/yql?q=select%20units,wind,atmosphere,astronomy,LOCATION%20from%20weather.forecast%20where%20woeid=551801%20AND%20u=%27c%27
                 Teil 2: http://query.yahooapis.com/v1/public/yql?q=select%20item%20from%20weather.forecast%20where%20woeid=551801%20AND%20u=%27c%27 *)

    	IF cycle = 0 THEN
      		URL_DATA.QUERY := 'q=select%20units,wind,atmosphere,astronomy,LOCATION%20from%20weather.forecast%20where%20woeid='; (* Teil 1 - infos *)
      	ELSE
      		URL_DATA.QUERY := 'q=select%20item%20from%20weather.forecast%20where%20woeid='; (* Teil 2 - Tagesdaten *)
      	END_IF

      	URL_DATA.QUERY := CONCAT(URL_DATA.QUERY,LOCATION); (* LOCATION *)

      	IF UNITS THEN
        		URL_DATA.QUERY := CONCAT(URL_DATA.QUERY,'%20and%20u=%27f%27'); (* fahrenheit *)
      	ELSE
        		URL_DATA.QUERY := CONCAT(URL_DATA.QUERY,'%20and%20u=%27c%27'); (* celsius *)
      	END_IF

      	URL_DATA.PATH := '/v1/public/yql';

      	state := 60;

    60:	IF HTTP_GET.DONE THEN
    		state := 80;
    		CTRL.START_POS := HTTP_GET.BODY_START;
    		CTRL.STOP_POS := HTTP_GET.BODY_STOP;
    		CTRL.COMMAND := WORD#2#10000000_00011000; (* ONLY TEXT AND ATTRIBUTE *)
    		CTRL.WATCHDOG  := T#1ms;

    	ELSIF (HTTP_GET.ERROR > DWORD#00) THEN
    		(* Fehlerbehandlung *)
    		ERROR_C := HTTP_GET.ERROR;
    		ERROR_T := BYTE#02;
    		state := 100;
    	END_IF

    80: XML_READER(CTRL:=CTRL,BUF:=R_BUF.BUFFER); (* XML Daten seriell lesen *)
    	IF CTRL.TYP < 98 THEN (* nur auswerten wenn kein Watchdog durchlauf *)
    		value_int := 0;
    		value_real := 0.0;
    		(* automatische konvertierung in real und int ausführen *)
    		IF LEN(CTRL.VALUE) <= 20 THEN
    			v_real:=FLOAT_TO_REAL(FLT:=CTRL.VALUE);
    			IF CHK_REAL(v_real) = 0 THEN (* !!! prüft auf gültigen REAL Wert, ansonsten kann Twincat 2.x abstürzen !!!!  *)
    				value_real := v_real;
    				value_int := REAL_TO_INT(value_real);
    			END_IF
    		END_IF

    		(*####################  DEBUG-MESSAGE  ###################################*)
    		(*IF _debug_enable THEN
    			LOG_CL.NEW_MSG := 'XML: ~2 # ~3 # ~4 # ~5';
    			LOG_CL.PRINTF[2] := UINT_TO_STRING(CTRL.LEVEL);
    			LOG_CL.PRINTF[3] := UINT_TO_STRING(CTRL.COUNT);
    			LOG_CL.PRINTF[4] := CTRL.ELEMENT;
    			LOG_CL.PRINTF[5] := CTRL.VALUE;
    			LOG_MSG();
    		END_IF*)
    		(*########################################################################*)

    		(* Antwortdaten stehen noch nicht bereit -> Warten und Abfrage wiederholen *)
    		IF CTRL.COUNT = 7 AND (CTRL.VALUE = '0')  THEN

    			repeat_count := repeat_count + USINT#1;

    			(* maximale Anzahl an Wiederholungen erreicht -> Mit Fehler abbrechen *)
    			IF repeat_count > repeat_max_count THEN

    				(* Fehlerbehandlung *)
    				ERROR_C := USINT_TO_DWORD(repeat_max_count);
    				ERROR_T := BYTE#03;
    				state   := 100;

    			ELSE
    				repeat_request := TRUE;
    				state := 100;

    				(*####################  DEBUG-MESSAGE  ###################################*)
    				(*IF _debug_enable THEN
    					LOG_CL.NEW_MSG := 'Request Error  / Part ~2 / Count ~3';
    					LOG_CL.PRINTF[2] := INT_TO_STRING(cycle);
    					LOG_CL.PRINTF[3] := USINT_TO_STRING(repeat_count);
    					LOG_MSG();
    				END_IF*)
    				(*########################################################################*)

    			END_IF

    		END_IF

    		IF cycle = 0 THEN
    	      		(* ------------ Teil 1 --------------*)
    	      		CASE UINT_TO_INT(CTRL.COUNT) OF
    	        		014: YW.location_city := CTRL.VALUE;
    	        		015: YW.location_country := CTRL.VALUE;
    	        		016: YW.location_region := CTRL.VALUE;
    	        		020: YW.wind_chill := value_int;
    	        		021: YW.wind_direction := value_int;
    	        		022: YW.wind_speed := value_real;
    	        		026: YW.atmosphere_humidity := value_int;
    	        		027: YW.atmosphere_pressure := value_real;
    	        		028: YW.atmosphere_rising := value_int;
    	        		029: YW.atmosphere_visibility := value_real;
    	        		033: YW.astronomy_sunrise := CTRL.VALUE;
    	        		034: YW.astronomy_sunset := CTRL.VALUE;
    	        		038: YW.unit_distance := CTRL.VALUE;
    	        		039: YW.unit_pressure := CTRL.VALUE;
    	        		040: YW.unit_speed := CTRL.VALUE;
    	        		041: YW.unit_temperature := CTRL.VALUE;
    	      		END_CASE
    	    	ELSE
    	      		(* ------------ Teil 2 --------------*)
    	      		CASE UINT_TO_INT(CTRL.COUNT) OF
    	        		018: YW.GEO_LATITUDE := value_real;
    	        		022: YW.GEO_LONGITUDE := value_real;

    			032: YW.CUR_CONDITIONS_CODE := value_int;
    			         YW.CUR_CONDITIONS_ICON := value_int;
    	        		034: YW.CUR_CONDITIONS_TEMP := value_int;
    	        		035: YW.CUR_CONDITIONS_TEXT := CTRL.VALUE;

    			039: YW.FORECAST_TODAY_CODE := value_int;
    			         YW.FORECAST_TODAY_ICON := value_int;
    			040: YW.FORECAST_TODAY_DATE_LONG := CTRL.VALUE;
    	        		042: YW.FORECAST_TODAY_HIGH_TEMP := value_int;
    	        		043: YW.FORECAST_TODAY_LOW_TEMP := value_int;
    	        		044: YW.FORECAST_TODAY_TEXT := CTRL.VALUE;

    			048..125: (* forcast day 1-10 *)
    				cnt := UINT_TO_INT(CTRL.COUNT) - 48;
    				day_idx := cnt / 9 + 1;
    				idx := cnt MOD 9;
    	      	  		CASE idx OF
    					0:	YW.FORECAST_DAY[day_idx].CODE := value_int;
    						YW.FORECAST_DAY[day_idx].ICON := value_int;
    					1:	YW.FORECAST_DAY[day_idx].DATE_LONG := CTRL.VALUE;
    					3:	YW.FORECAST_DAY[day_idx].HIGH_TEMP := value_int;
    					4:	YW.FORECAST_DAY[day_idx].LOW_TEMP := value_int;
    					5:	YW.FORECAST_DAY[day_idx].TEXT := CTRL.VALUE;
    	      	  		END_CASE
    	      		END_CASE
    	    	END_IF
    	ELSIF CTRL.TYP = 99 THEN (* EXIT - letztes Element gelesen *)
    		state := 100;
    	END_IF

    100:	(* UNLOCK HTTP DATA *)
    	IF (NOT HTTP_GET.DONE) THEN

    		IF repeat_request THEN
    			repeat_tx := tx;
        			state := 110;

    		ELSIF cycle = 0 AND ERROR_T = BYTE#0 THEN
    			(* Teil 2 ausführen *)
        			state := 50;
    			cycle := cycle + 1;
    			repeat_count := USINT#0;
    		ELSE
    	    		state := 0;
    	    		BUSY  := FALSE;
    	    		DONE := ERROR_T = BYTE#0;
    		END_IF
    	END_IF

    110: (* REPEAT REQUEST - WAIT TIME *)
    	IF tx > repeat_tx + repeat_wait_time THEN

    		(*####################  DEBUG-MESSAGE  ###################################*)
    		(*IF _debug_enable THEN
    			LOG_CL.NEW_MSG := 'Repeat request after waittime / Part ~2 / Count ~3';
    			LOG_CL.PRINTF[2] := INT_TO_STRING(cycle);
    			LOG_CL.PRINTF[3] := USINT_TO_STRING(repeat_count);
    			LOG_MSG();
    		END_IF*)
    		(*########################################################################*)

    		repeat_request := FALSE;
    		state := 50;

    	END_IF

    END_CASE

    (* ---------------- DNS --------------- *)
    DNS_CLIENT(	IP_C:=IP_C,
    			S_BUF:=S_BUF,
    			R_BUF:=R_BUF,
    			DOMAIN:=URL_DATA.DOMAIN,
    			IP4_DNS:=DWORD#00,
    			ACTIVATE:=state=40 (* DNS Start *)
    			);
    (* nicht oder nicht direkt verwendete Parameter *)
    (*	DWORD :=DNS_CLIENT.IP4;
    	BOOL  :=DNS_CLIENT.DONE;
    	BYTE  :=DNS_CLIENT.ERROR; *)
    (* -------------------------------------*)

    (* ------------- HTTP_GET --------------- *)
    HTTP_GET(	IP_C:=IP_C,
    			S_BUF:=S_BUF,
    			R_BUF:=R_BUF,
    			IP4:=DNS_CLIENT.IP4,
    			GET:=state=60,
    			MODE:=BYTE#2, (* HTTP 1.1 mit persistenter Verbindung *)
    			UNLOCK_BUF:=state=100,
    			URL_DATA:=URL_DATA
    			);

    (* nicht oder nicht direkt verwendete Parameter *)
    (*	STRING := HTTP_GET.HTTP_STATUS;
    	UINT :=HTTP_GET.HEADER_START;
    	UINT :=HTTP_GET.HEADER_STOP;
    	UINT :=HTTP_GET.BODY_START;
    	UINT :=HTTP_GET.BODY_STOP;
    	BOOL :=HTTP_GET.DONE;
    	BYTE :=HTTP_GET.ERROR;
    *)
    (* -------------------------------------*)

    activate_last := ACTIVATE;

    (*####################  DEBUG-MESSAGE  ###################################*)
    (*IF _debug_enable THEN
    	IF state <> _debug_state_last THEN
    		LOG_CL.NEW_MSG := 'YW-step: /last ~1 /New ~2';
    		LOG_CL.PRINTF[1] := INT_TO_STRING(_debug_state_last);
    		LOG_CL.PRINTF[2] := INT_TO_STRING(state);
    		LOG_MSG();
    		_debug_state_last := state;
    	END_IF
    END_IF*)
    (*########################################################################*)

    (* revision history
    ks	18. dez. 2008	rev 1.0
    	original version

    ks	01. oct. 2009	rev 1.1
    	YAHOO_WEATHER_DATA

    ks	24. sep. 2010	rev 1.2
    	new URL-LOCATION-parameter and REAL_CHECK (TwinCat BUG)

    ks	04. may. 2011	rev 1.3
    	neue elemente:  CUR_CONDITIONS_ICON, FORCAST_TODAY_ICON, FORCAST_TOMORROW_ICON

    ks	30. mar. 2016	rev 1.4
    	änderung der api schnittstelle (URL) von yahoo

    ks	01. jun. 2016	rev 1.5
    	komplette überarbeitung auf neue yahoo-api

    ks	22. may. 2017	rev 1.6
    	automatische wiederholung der Abfrage wenn keine Daten vorhanden sind
    *)
END_FUNCTION_BLOCK

(* ---- YAHOO_WEATHER_DESC_GE.st ---- *)
FUNCTION_BLOCK YAHOO_WEATHER_DESC_GE
    (*http://www.oscat.de/images/OSCATBasic/oscat_basic333_en.pdf#page=214*)
    IF ACTIVATE AND act_last = FALSE THEN
    	FOR y := 1 TO 12 DO
    		CASE y OF
    		01:	x := YW.CUR_CONDITIONS_CODE;

    		02:	YW.CUR_CONDITIONS_TEXT := str;
    			x := YW.FORECAST_TODAY_CODE;
    		03:	YW.FORECAST_TODAY_TEXT := str;
    			x := YW.FORECAST_DAY[1].CODE;
    		04:	YW.FORECAST_DAY[1].TEXT := str;
    			x := YW.FORECAST_DAY[2].CODE;
    		05:	YW.FORECAST_DAY[2].TEXT := str;
    			x := YW.FORECAST_DAY[3].CODE;
    		06:	YW.FORECAST_DAY[3].TEXT := str;
    			x := YW.FORECAST_DAY[4].CODE;
    		07:	YW.FORECAST_DAY[4].TEXT := str;
    			x := YW.FORECAST_DAY[5].CODE;
    		08:	YW.FORECAST_DAY[5].TEXT := str;
    			x := YW.FORECAST_DAY[6].CODE;
    		09:	YW.FORECAST_DAY[6].TEXT := str;
    			x := YW.FORECAST_DAY[7].CODE;
    		10:	YW.FORECAST_DAY[7].TEXT := str;
    			x := YW.FORECAST_DAY[8].CODE;
    		11:	YW.FORECAST_DAY[8].TEXT := str;
    			x := YW.FORECAST_DAY[9].CODE;
    		12:	YW.FORECAST_DAY[9].TEXT := str;
    		END_CASE

    		CASE x OF
    		00:	str := 'Wirbelsturm';
    		01:	str := 'Tropensturm';
    		02:	str := 'Wirbelsturm';
    		03:	str := 'starkes Gewitter ';
    		04:	str := 'Gewitter';
    		05:	str := 'Schneeregen';
    		06:	str := 'Schneeregen';
    		07:	str := 'Schneeregen';
    		08:	str := 'gefrierender Nieselregen';
    		09:	str := 'Nieselregen';
    		10:	str := 'gefrierender Regen';
    		11:	str := 'Regenfälle';
    		12:	str := 'Regenfälle';
    		13:	str := 'Schneegestöber';
    		14:	str := 'leichte Schneefälle';
    		15:	str := 'Schneetreiben';
    		16:	str := 'Schnee';
    		17:	str := 'Hagel';
    		18:	str := 'Schneeregen';
    		19:	str := 'Staub';
    		20:	str := 'nebelig';
    		21:	str := 'Dunst';
    		22:	str := 'rauchig';
    		23:	str := 'stürmisch';
    		24:	str := 'windig';
    		25:	str := 'kalt';
    		26:	str := 'bewölkt';
    		27:	str := 'meist bewölkt';
    		28:	str := 'meist bewölkt';
    		29:	str := 'teilweise bewölkt';
    		30:	str := 'teilweise bewölkt';
    		31:	str := 'klar';
    		32:	str := 'sonnig';
    		33:	str := 'heiter';
    		34:	str := 'heiter';
    		35:	str := 'Regen und Hagel';
    		36:	str := 'heiß';
    		37:	str := 'örtliche Gewitter';
    		38:	str := 'vereinzelte Gewitter';
    		39:	str := 'vereinzelte Gewitter';
    		40:	str := 'vereinzelte Regenfälle';
    		41:	str := 'schwere Schneefälle';
    		42:	str := 'vereinzelte Schneefälle';
    		43:	str := 'schwere Schneefälle';
    		44:	str := 'teilweise bewölkt';
    		45:	str := 'gewittrige Regenfälle';
    		46:	str := 'Schneefälle';
    		47:	str := 'örtliche gewittrige Regenfälle';
    		ELSE
    			str := 'nicht verfügbar';
    		END_CASE
    	END_FOR
    END_IF
    act_last := ACTIVATE;

    (* revision history
    ks	04. may. 2011	rev 1.0
    	original version
    ks	01. jun. 2016	rev 1.1
    	komplette überarbeitung auf neue yahoo-api

    *)
END_FUNCTION_BLOCK

(* ---- YAHOO_WEATHER_ICON_OSCAT.st ---- *)
FUNCTION_BLOCK YAHOO_WEATHER_ICON_OSCAT
    (*http://www.oscat.de/images/OSCATNetwork/oscat_netlib121_en.pdf#page=211*)
    IF ACTIVATE AND act_last = FALSE THEN
    	x := MIN(YW.CUR_CONDITIONS_CODE,48);
    	YW.CUR_CONDITIONS_ICON := dat[x];
    	x := MIN(YW.FORECAST_TODAY_CODE,48);
    	YW.FORECAST_TODAY_ICON := dat[x];
    	FOR idx := 1 TO 9 DO
    		x := MIN(YW.FORECAST_DAY[idx].CODE,48);
    		YW.FORECAST_DAY[idx].ICON := dat[x];
    	END_FOR
    END_IF
    act_last := ACTIVATE;

    (* revision history
    ks	04. may. 2011	rev 1.0
    	original version

    ks	01. jun. 2016	rev 1.1
    	komplette überarbeitung auf neue yahoo-api
    *)
END_FUNCTION_BLOCK

(* ---- oscatNetw.var ---- *)
VAR CONSTANT
END_VAR
